LIN {X 0,Y 418.264,Z 439.007,A -85,B 0,C 180,E1 -10279.791,E2 -10279.791} C_VEL
LIN {X 0,Y 418.232,Z 439.016,A -85,B 0,C 180,E1 -10282.737,E2 -10282.737} C_VEL
LIN {X 0,Y 418.265,Z 439.008,A -85,B 0,C 180,E1 -10285.905,E2 -10285.905} C_VEL
LIN {X 0,Y 418.269,Z 439.007,A -85,B 0,C 180,E1 -10289.162,E2 -10289.162} C_VEL
LIN {X 0,Y 418.255,Z 439.008,A -85,B 0,C 180,E1 -10292.845,E2 -10292.845} C_VEL
LIN {X 0,Y 418.245,Z 439.015,A -85,B 0,C 180,E1 -10296.24,E2 -10296.24} C_VEL
LIN {X 0,Y 418.277,Z 439.018,A -85,B 0,C 180,E1 -10298.25,E2 -10298.25} C_VEL
LIN {X 0,Y 421.028,Z 450.162,A -85,B 0,C 180,E1 -10300.737,E2 -10300.737} C_VEL
LIN {X 0,Y 429.428,Z 469.629,A -85,B 0,C 180,E1 -10301.712,E2 -10301.712} C_VEL
LIN {X 0,Y 431.13,Z 477.405,A -85,B 0,C 180,E1 -10301.972,E2 -10301.972} C_VEL
LIN {X 0,Y 428.557,Z 614.749,A -85,B 0,C 180,E1 -10304.367,E2 -10304.367} C_VEL
LIN {X 0,Y 427.904,Z 630.406,A -85,B 0,C 180,E1 -10304.826,E2 -10304.826} C_VEL
LIN {X 0,Y 427.072,Z 645.206,A -85,B 0,C 180,E1 -10305.458,E2 -10305.458} C_VEL
LIN {X 0,Y 426.047,Z 660.031,A -85,B 0,C 180,E1 -10306.303,E2 -10306.303} C_VEL
LIN {X 0,Y 424.862,Z 673.816,A -85,B 0,C 180,E1 -10307.297,E2 -10307.297} C_VEL
LIN {X 0,Y 423.692,Z 686.587,A -85,B 0,C 180,E1 -10308.434,E2 -10308.434} C_VEL
LIN {X 0,Y 422.369,Z 699.367,A -85,B 0,C 180,E1 -10309.814,E2 -10309.814} C_VEL
LIN {X 0,Y 421.205,Z 710.398,A -85,B 0,C 180,E1 -10311.252,E2 -10311.252} C_VEL
LIN {X 0,Y 420.173,Z 719.587,A -85,B 0,C 180,E1 -10312.676,E2 -10312.676} C_VEL
LIN {X 0,Y 419.262,Z 728.801,A -85,B 0,C 180,E1 -10314.374,E2 -10314.374} C_VEL
LIN {X 0,Y 418.549,Z 736.533,A -85,B 0,C 180,E1 -10316.09,E2 -10316.09} C_VEL
LIN {X 0,Y 417.858,Z 743.619,A -85,B 0,C 180,E1 -10318.009,E2 -10318.009} C_VEL
LIN {X 0,Y 417.543,Z 748.582,A -85,B 0,C 180,E1 -10319.673,E2 -10319.673} C_VEL
LIN {X 0,Y 417.249,Z 752.105,A -85,B 0,C 180,E1 -10321.149,E2 -10321.149} C_VEL
LIN {X 0,Y 416.99,Z 755.939,A -85,B 0,C 180,E1 -10323.288,E2 -10323.288} C_VEL
LIN {X 0,Y 416.875,Z 758.426,A -85,B 0,C 180,E1 -10325.558,E2 -10325.558} C_VEL
LIN {X 0,Y 416.837,Z 759.366,A -85,B 0,C 180,E1 -10328.021,E2 -10328.021} C_VEL
LIN {X 0,Y 416.862,Z 758.566,A -85,B 0,C 180,E1 -10330.295,E2 -10330.295} C_VEL
LIN {X 0,Y 416.983,Z 756.515,A -85,B 0,C 180,E1 -10332.34,E2 -10332.34} C_VEL
LIN {X 0,Y 417.189,Z 753.759,A -85,B 0,C 180,E1 -10334.039,E2 -10334.039} C_VEL
LIN {X 0,Y 416.614,Z 752.269,A -85,B 0,C 180,E1 -10334.821,E2 -10334.821} C_VEL
LIN {X 0,Y 413.918,Z 749.553,A -85,B 0,C 180,E1 -10336.084,E2 -10336.084} C_VEL
LIN {X 0,Y 411.683,Z 747.027,A -85,B 0,C 180,E1 -10337.087,E2 -10337.087} C_VEL
LIN {X 0,Y 410.83,Z 744.837,A -85,B 0,C 180,E1 -10337.846,E2 -10337.846} C_VEL
LIN {X 0,Y 410.82,Z 744.026,A -85,B 0,C 180,E1 -10338.098,E2 -10338.098} C_VEL
LIN {X 0,Y 411.441,Z 736.535,A -85,B 0,C 180,E1 -10340.166,E2 -10340.166} C_VEL
LIN {X 0,Y 412.264,Z 728.503,A -85,B 0,C 180,E1 -10341.956,E2 -10341.956} C_VEL
LIN {X 0,Y 413.238,Z 719.329,A -85,B 0,C 180,E1 -10343.654,E2 -10343.654} C_VEL
LIN {X 0,Y 414.315,Z 709.798,A -85,B 0,C 180,E1 -10345.135,E2 -10345.135} C_VEL
LIN {X 0,Y 415.491,Z 698.732,A -85,B 0,C 180,E1 -10346.583,E2 -10346.583} C_VEL
LIN {X 0,Y 416.83,Z 686.135,A -85,B 0,C 180,E1 -10347.947,E2 -10347.947} C_VEL
LIN {X 0,Y 418.019,Z 674.003,A -85,B 0,C 180,E1 -10349.037,E2 -10349.037} C_VEL
LIN {X 0,Y 419.145,Z 660.909,A -85,B 0,C 180,E1 -10350.001,E2 -10350.001} C_VEL
LIN {X 0,Y 420.189,Z 646.609,A -85,B 0,C 180,E1 -10350.839,E2 -10350.839} C_VEL
LIN {X 0,Y 421.045,Z 631.881,A -85,B 0,C 180,E1 -10351.495,E2 -10351.495} C_VEL
LIN {X 0,Y 421.681,Z 616.76,A -85,B 0,C 180,E1 -10351.97,E2 -10351.97} C_VEL
LIN {X 0,Y 422.249,Z 590.391,A -85,B 0,C 180,E1 -10352.469,E2 -10352.469} C_VEL
LIN {X 0,Y 424.329,Z 477.84,A -85,B 0,C 180,E1 -10354.433,E2 -10354.433} C_VEL
LIN {X 0,Y 422.249,Z 469.646,A -85,B 0,C 180,E1 -10354.725,E2 -10354.725} C_VEL
LIN {X 0,Y 413.752,Z 449.749,A -85,B 0,C 180,E1 -10355.705,E2 -10355.705} C_VEL
LIN {X 0,Y 411.414,Z 439.866,A -85,B 0,C 180,E1 -10357.917,E2 -10357.917} C_VEL
LIN {X 0,Y 411.303,Z 439.874,A -85,B 0,C 180,E1 -10361.833,E2 -10361.833} C_VEL
LIN {X 0,Y 411.267,Z 439.881,A -85,B 0,C 180,E1 -10364.853,E2 -10364.853} C_VEL
LIN {X 0,Y 411.257,Z 439.88,A -85,B 0,C 180,E1 -10367.915,E2 -10367.915} C_VEL
LIN {X 0,Y 411.206,Z 439.885,A -85,B 0,C 180,E1 -10371.034,E2 -10371.034} C_VEL
LIN {X 0,Y 411.231,Z 439.879,A -85,B 0,C 180,E1 -10374.215,E2 -10374.215} C_VEL
LIN {X 0,Y 411.263,Z 439.878,A -85,B 0,C 180,E1 -10377.478,E2 -10377.478} C_VEL
LIN {X 0,Y 411.2,Z 439.888,A -85,B 0,C 180,E1 -10380.847,E2 -10380.847} C_VEL
LIN {X 0,Y 411.21,Z 439.886,A -85,B 0,C 180,E1 -10384.333,E2 -10384.333} C_VEL
LIN {X 0,Y 411.204,Z 439.879,A -85,B 0,C 180,E1 -10387.973,E2 -10387.973} C_VEL
LIN {X 0,Y 411.197,Z 439.889,A -85,B 0,C 180,E1 -10391.233,E2 -10391.233} C_VEL
LIN {X 0,Y 411.182,Z 439.887,A -85,B 0,C 180,E1 -10394.49,E2 -10394.49} C_VEL
LIN {X 0,Y 411.201,Z 439.879,A -85,B 0,C 180,E1 -10398.197,E2 -10398.197} C_VEL
LIN {X 0,Y 411.232,Z 439.882,A -85,B 0,C 180,E1 -10400.777,E2 -10400.777} C_VEL
LIN {X 0,Y 411.202,Z 439.879,A -85,B 0,C 180,E1 -10404.471,E2 -10404.471} C_VEL
LIN {X 0,Y 411.209,Z 439.885,A -85,B 0,C 180,E1 -10406.873,E2 -10406.873} C_VEL
LIN {X 0,Y 411.234,Z 439.873,A -85,B 0,C 180,E1 -10410.644,E2 -10410.644} C_VEL
LIN {X 0,Y 411.239,Z 439.888,A -85,B 0,C 180,E1 -10413.619,E2 -10413.619} C_VEL
LIN {X 0,Y 411.198,Z 439.874,A -85,B 0,C 180,E1 -10416.852,E2 -10416.852} C_VEL
LIN {X 0,Y 411.216,Z 439.886,A -85,B 0,C 180,E1 -10420.05,E2 -10420.05} C_VEL
LIN {X 0,Y 411.264,Z 439.871,A -85,B 0,C 180,E1 -10423.131,E2 -10423.131} C_VEL
LIN {X 0,Y 411.306,Z 439.872,A -85,B 0,C 180,E1 -10426.896,E2 -10426.896} C_VEL
LIN {X 0,Y 411.293,Z 439.865,A -85,B 0,C 180,E1 -10430.161,E2 -10430.161} C_VEL
LIN {X 0,Y 411.482,Z 439.851,A -85,B 0,C 180,E1 -10432.146,E2 -10432.146} C_VEL
LIN {X 0,Y 411.475,Z 439.853,A -85,B 0,C 180,E1 -10434.118,E2 -10434.118} C_VEL
LIN {X 0,Y 411.511,Z 439.845,A -85,B 0,C 180,E1 -10438.042,E2 -10438.042} C_VEL
LIN {X 0,Y 411.642,Z 439.835,A -85,B 0,C 180,E1 -10440,E2 -10440} C_VEL
LIN {X 0,Y 411.466,Z 439.848,A -85,B 0,C 180,E1 -10442.937,E2 -10442.937} C_VEL
LIN {X 0,Y 411.46,Z 439.85,A -85,B 0,C 180,E1 -10446.867,E2 -10446.867} C_VEL
LIN {X 0,Y 411.354,Z 439.867,A -85,B 0,C 180,E1 -10448.845,E2 -10448.845} C_VEL
LIN {X 0,Y 411.283,Z 439.866,A -85,B 0,C 180,E1 -10451.833,E2 -10451.833} C_VEL
LIN {X 0,Y 411.26,Z 439.878,A -85,B 0,C 180,E1 -10454.852,E2 -10454.852} C_VEL
LIN {X 0,Y 411.252,Z 439.871,A -85,B 0,C 180,E1 -10457.915,E2 -10457.915} C_VEL
LIN {X 0,Y 411.196,Z 439.886,A -85,B 0,C 180,E1 -10461.034,E2 -10461.034} C_VEL
LIN {X 0,Y 411.227,Z 439.885,A -85,B 0,C 180,E1 -10464.215,E2 -10464.215} C_VEL
LIN {X 0,Y 411.259,Z 439.883,A -85,B 0,C 180,E1 -10467.477,E2 -10467.477} C_VEL
LIN {X 0,Y 411.196,Z 439.885,A -85,B 0,C 180,E1 -10470.847,E2 -10470.847} C_VEL
LIN {X 0,Y 411.206,Z 439.887,A -85,B 0,C 180,E1 -10474.333,E2 -10474.333} C_VEL
LIN {X 0,Y 411.201,Z 439.889,A -85,B 0,C 180,E1 -10477.973,E2 -10477.973} C_VEL
LIN {X 0,Y 411.183,Z 439.889,A -85,B 0,C 180,E1 -10480.504,E2 -10480.504} C_VEL
LIN {X 0,Y 411.175,Z 439.891,A -85,B 0,C 180,E1 -10483.133,E2 -10483.133} C_VEL
LIN {X 0,Y 411.227,Z 439.886,A -85,B 0,C 180,E1 -10485.872,E2 -10485.872} C_VEL
LIN {X 0,Y 411.205,Z 439.888,A -85,B 0,C 180,E1 -10488.765,E2 -10488.765} C_VEL
LIN {X 0,Y 411.194,Z 439.892,A -85,B 0,C 180,E1 -10492.026,E2 -10492.026} C_VEL
LIN {X 0,Y 411.206,Z 439.887,A -85,B 0,C 180,E1 -10495.666,E2 -10495.666} C_VEL
LIN {X 0,Y 411.206,Z 439.954,A -85,B 0,C 180,E1 -10496.552,E2 -10496.552} C_VEL
LIN {X 0,Y 415.186,Z 455.473,A -85,B 0,C 180,E1 -10499.688,E2 -10499.688} C_VEL
LIN {X 0,Y 417.73,Z 467.012,A -85,B 0,C 180,E1 -10501.895,E2 -10501.895} C_VEL
LIN {X 0,Y 417.421,Z 471.137,A -85,B 0,C 180,E1 -10502.59,E2 -10502.59} C_VEL
LIN {X 0,Y 423.956,Z 504.652,A -85,B 0,C 180,E1 -10503.663,E2 -10503.663} C_VEL
LIN {X 0,Y 422.062,Z 609.761,A -85,B 0,C 180,E1 -10505.498,E2 -10505.498} C_VEL
LIN {X 0,Y 421.485,Z 639.304,A -85,B 0,C 180,E1 -10506.051,E2 -10506.051} C_VEL
LIN {X 0,Y 420.701,Z 654.425,A -85,B 0,C 180,E1 -10506.512,E2 -10506.512} C_VEL
LIN {X 0,Y 419.794,Z 669.444,A -85,B 0,C 180,E1 -10507.175,E2 -10507.175} C_VEL
LIN {X 0,Y 418.751,Z 682.833,A -85,B 0,C 180,E1 -10507.943,E2 -10507.943} C_VEL
LIN {X 0,Y 417.533,Z 696.274,A -85,B 0,C 180,E1 -10508.912,E2 -10508.912} C_VEL
LIN {X 0,Y 416.123,Z 709.958,A -85,B 0,C 180,E1 -10510.129,E2 -10510.129} C_VEL
LIN {X 0,Y 414.772,Z 722.886,A -85,B 0,C 180,E1 -10511.541,E2 -10511.541} C_VEL
LIN {X 0,Y 413.69,Z 733.682,A -85,B 0,C 180,E1 -10512.959,E2 -10512.959} C_VEL
LIN {X 0,Y 412.496,Z 744.676,A -85,B 0,C 180,E1 -10514.687,E2 -10514.687} C_VEL
LIN {X 0,Y 411.586,Z 753.834,A -85,B 0,C 180,E1 -10516.428,E2 -10516.428} C_VEL
LIN {X 0,Y 411.006,Z 761.372,A -85,B 0,C 180,E1 -10518.159,E2 -10518.159} C_VEL
LIN {X 0,Y 410.407,Z 768.44,A -85,B 0,C 180,E1 -10520.139,E2 -10520.139} C_VEL
LIN {X 0,Y 410.156,Z 774.002,A -85,B 0,C 180,E1 -10522.121,E2 -10522.121} C_VEL
LIN {X 0,Y 409.975,Z 778.206,A -85,B 0,C 180,E1 -10524.096,E2 -10524.096} C_VEL
LIN {X 0,Y 409.895,Z 781.155,A -85,B 0,C 180,E1 -10526.067,E2 -10526.067} C_VEL
LIN {X 0,Y 409.957,Z 782.918,A -85,B 0,C 180,E1 -10528.035,E2 -10528.035} C_VEL
LIN {X 0,Y 409.923,Z 783.517,A -85,B 0,C 180,E1 -10529.999,E2 -10529.999} C_VEL
LIN {X 0,Y 409.959,Z 782.915,A -85,B 0,C 180,E1 -10531.964,E2 -10531.964} C_VEL
LIN {X 0,Y 409.907,Z 781.16,A -85,B 0,C 180,E1 -10533.932,E2 -10533.932} C_VEL
LIN {X 0,Y 409.976,Z 778.229,A -85,B 0,C 180,E1 -10535.903,E2 -10535.903} C_VEL
LIN {X 0,Y 410.155,Z 774.051,A -85,B 0,C 180,E1 -10537.878,E2 -10537.878} C_VEL
LIN {X 0,Y 410.407,Z 768.515,A -85,B 0,C 180,E1 -10539.86,E2 -10539.86} C_VEL
LIN {X 0,Y 411.027,Z 761.48,A -85,B 0,C 180,E1 -10541.84,E2 -10541.84} C_VEL
LIN {X 0,Y 411.627,Z 753.862,A -85,B 0,C 180,E1 -10543.596,E2 -10543.596} C_VEL
LIN {X 0,Y 412.489,Z 744.879,A -85,B 0,C 180,E1 -10545.312,E2 -10545.312} C_VEL
LIN {X 0,Y 413.694,Z 733.993,A -85,B 0,C 180,E1 -10547.04,E2 -10547.04} C_VEL
LIN {X 0,Y 414.994,Z 722.266,A -85,B 0,C 180,E1 -10548.581,E2 -10548.581} C_VEL
LIN {X 0,Y 416.161,Z 710.536,A -85,B 0,C 180,E1 -10549.868,E2 -10549.868} C_VEL
LIN {X 0,Y 417.546,Z 697.077,A -85,B 0,C 180,E1 -10551.086,E2 -10551.086} C_VEL
LIN {X 0,Y 418.806,Z 683.881,A -85,B 0,C 180,E1 -10552.053,E2 -10552.053} C_VEL
LIN {X 0,Y 419.957,Z 669.116,A -85,B 0,C 180,E1 -10552.918,E2 -10552.918} C_VEL
LIN {X 0,Y 420.932,Z 654.325,A -85,B 0,C 180,E1 -10553.57,E2 -10553.57} C_VEL
LIN {X 0,Y 421.717,Z 639.333,A -85,B 0,C 180,E1 -10554.032,E2 -10554.032} C_VEL
LIN {X 0,Y 422.307,Z 613.685,A -85,B 0,C 180,E1 -10554.519,E2 -10554.519} C_VEL
LIN {X 0,Y 424.314,Z 504.605,A -85,B 0,C 180,E1 -10556.434,E2 -10556.434} C_VEL
LIN {X 0,Y 419.497,Z 479.497,A -85,B 0,C 180,E1 -10557.255,E2 -10557.255} C_VEL
LIN {X 0,Y 417.605,Z 470.44,A -85,B 0,C 180,E1 -10557.594,E2 -10557.594} C_VEL
LIN {X 0,Y 417.693,Z 466.142,A -85,B 0,C 180,E1 -10558.343,E2 -10558.343} C_VEL
LIN {X 0,Y 414.395,Z 451.915,A -85,B 0,C 180,E1 -10561.148,E2 -10561.148} C_VEL
LIN {X 0,Y 411.222,Z 439.886,A -85,B 0,C 180,E1 -10563.703,E2 -10563.703} C_VEL
LIN {X 0,Y 411.189,Z 439.89,A -85,B 0,C 180,E1 -10566.741,E2 -10566.741} C_VEL
LIN {X 0,Y 411.224,Z 439.882,A -85,B 0,C 180,E1 -10569.73,E2 -10569.73} C_VEL
LIN {X 0,Y 411.217,Z 439.881,A -85,B 0,C 180,E1 -10573.127,E2 -10573.127} C_VEL
LIN {X 0,Y 411.166,Z 439.891,A -85,B 0,C 180,E1 -10575.88,E2 -10575.88} C_VEL
LIN {X 0,Y 411.159,Z 439.895,A -85,B 0,C 180,E1 -10578.771,E2 -10578.771} C_VEL
LIN {X 0,Y 411.205,Z 439.888,A -85,B 0,C 180,E1 -10581.83,E2 -10581.83} C_VEL
LIN {X 0,Y 411.205,Z 439.887,A -85,B 0,C 180,E1 -10585.121,E2 -10585.121} C_VEL
LIN {X 0,Y 411.159,Z 439.893,A -85,B 0,C 180,E1 -10588.002,E2 -10588.002} C_VEL
LIN {X 0,Y 411.211,Z 439.886,A -85,B 0,C 180,E1 -10591.41,E2 -10591.41} C_VEL
LIN {X 0,Y 411.231,Z 439.88,A -85,B 0,C 180,E1 -10593.619,E2 -10593.619} C_VEL
LIN {X 0,Y 411.196,Z 439.889,A -85,B 0,C 180,E1 -10596.852,E2 -10596.852} C_VEL
LIN {X 0,Y 411.207,Z 439.884,A -85,B 0,C 180,E1 -10600.05,E2 -10600.05} C_VEL
LIN {X 0,Y 411.255,Z 439.875,A -85,B 0,C 180,E1 -10603.131,E2 -10603.131} C_VEL
LIN {X 0,Y 411.306,Z 439.871,A -85,B 0,C 180,E1 -10606.891,E2 -10606.891} C_VEL
LIN {X 0,Y 411.301,Z 439.874,A -85,B 0,C 180,E1 -10610.162,E2 -10610.162} C_VEL
LIN {X 0,Y 411.453,Z 439.853,A -85,B 0,C 180,E1 -10613.133,E2 -10613.133} C_VEL
LIN {X 0,Y 411.306,Z 439.873,A -85,B 0,C 180,E1 -10615.099,E2 -10615.099} C_VEL
LIN {X 0,Y 411.507,Z 439.846,A -85,B 0,C 180,E1 -10618.043,E2 -10618.043} C_VEL
LIN {X 0,Y 411.634,Z 439.836,A -85,B 0,C 180,E1 -10620,E2 -10620} C_VEL
LIN {X 0,Y 411.46,Z 439.856,A -85,B 0,C 180,E1 -10622.937,E2 -10622.937} C_VEL
LIN {X 0,Y 411.454,Z 439.856,A -85,B 0,C 180,E1 -10626.867,E2 -10626.867} C_VEL
LIN {X 0,Y 411.286,Z 439.878,A -85,B 0,C 180,E1 -10629.839,E2 -10629.839} C_VEL
LIN {X 0,Y 411.298,Z 439.874,A -85,B 0,C 180,E1 -10633.105,E2 -10633.105} C_VEL
LIN {X 0,Y 411.257,Z 439.882,A -85,B 0,C 180,E1 -10635.868,E2 -10635.868} C_VEL
LIN {X 0,Y 411.218,Z 439.885,A -85,B 0,C 180,E1 -10638.949,E2 -10638.949} C_VEL
LIN {X 0,Y 411.198,Z 439.894,A -85,B 0,C 180,E1 -10642.643,E2 -10642.643} C_VEL
LIN {X 0,Y 411.231,Z 439.886,A -85,B 0,C 180,E1 -10645.294,E2 -10645.294} C_VEL
LIN {X 0,Y 411.219,Z 439.89,A -85,B 0,C 180,E1 -10648.59,E2 -10648.59} C_VEL
LIN {X 0,Y 411.166,Z 439.893,A -85,B 0,C 180,E1 -10651.998,E2 -10651.998} C_VEL
LIN {X 0,Y 411.196,Z 439.891,A -85,B 0,C 180,E1 -10655.529,E2 -10655.529} C_VEL
LIN {X 0,Y 411.232,Z 439.979,A -85,B 0,C 180,E1 -10657.815,E2 -10657.815} C_VEL
LIN {X 0,Y 413.902,Z 450.487,A -85,B 0,C 180,E1 -10660.216,E2 -10660.216} C_VEL
LIN {X 0,Y 423.271,Z 471.849,A -85,B 0,C 180,E1 -10661.324,E2 -10661.324} C_VEL
LIN {X 0,Y 424.816,Z 478.598,A -85,B 0,C 180,E1 -10661.562,E2 -10661.562} C_VEL
LIN {X 0,Y 422.093,Z 615.228,A -85,B 0,C 180,E1 -10663.979,E2 -10663.979} C_VEL
LIN {X 0,Y 421.427,Z 630.771,A -85,B 0,C 180,E1 -10664.446,E2 -10664.446} C_VEL
LIN {X 0,Y 420.524,Z 645.75,A -85,B 0,C 180,E1 -10665.096,E2 -10665.096} C_VEL
LIN {X 0,Y 419.504,Z 659.931,A -85,B 0,C 180,E1 -10665.915,E2 -10665.915} C_VEL
LIN {X 0,Y 418.246,Z 674.101,A -85,B 0,C 180,E1 -10666.951,E2 -10666.951} C_VEL
LIN {X 0,Y 417,Z 686.839,A -85,B 0,C 180,E1 -10668.102,E2 -10668.102} C_VEL
LIN {X 0,Y 415.665,Z 699.15,A -85,B 0,C 180,E1 -10669.449,E2 -10669.449} C_VEL
LIN {X 0,Y 414.504,Z 709.69,A -85,B 0,C 180,E1 -10670.834,E2 -10670.834} C_VEL
LIN {X 0,Y 413.254,Z 720.367,A -85,B 0,C 180,E1 -10672.504,E2 -10672.504} C_VEL
LIN {X 0,Y 412.246,Z 729.718,A -85,B 0,C 180,E1 -10674.276,E2 -10674.276} C_VEL
LIN {X 0,Y 411.516,Z 737.209,A -85,B 0,C 180,E1 -10675.993,E2 -10675.993} C_VEL
LIN {X 0,Y 410.806,Z 744.291,A -85,B 0,C 180,E1 -10677.972,E2 -10677.972} C_VEL
LIN {X 0,Y 410.46,Z 749.144,A -85,B 0,C 180,E1 -10679.663,E2 -10679.663} C_VEL
LIN {X 0,Y 410.052,Z 754.007,A -85,B 0,C 180,E1 -10681.88,E2 -10681.88} C_VEL
LIN {X 0,Y 409.882,Z 756.625,A -85,B 0,C 180,E1 -10683.526,E2 -10683.526} C_VEL
LIN {X 0,Y 409.776,Z 758.784,A -85,B 0,C 180,E1 -10685.694,E2 -10685.694} C_VEL
LIN {X 0,Y 409.727,Z 759.555,A -85,B 0,C 180,E1 -10687.859,E2 -10687.859} C_VEL
LIN {X 0,Y 409.756,Z 758.996,A -85,B 0,C 180,E1 -10689.939,E2 -10689.939} C_VEL
LIN {X 0,Y 409.855,Z 757.165,A -85,B 0,C 180,E1 -10692.023,E2 -10692.023} C_VEL
LIN {X 0,Y 410.12,Z 754.049,A -85,B 0,C 180,E1 -10694.087,E2 -10694.087} C_VEL
LIN {X 0,Y 410.409,Z 749.635,A -85,B 0,C 180,E1 -10696.129,E2 -10696.129} C_VEL
LIN {X 0,Y 410.82,Z 744.026,A -85,B 0,C 180,E1 -10698.098,E2 -10698.098} C_VEL
LIN {X 0,Y 410.391,Z 741.613,A -85,B 0,C 180,E1 -10698.847,E2 -10698.847} C_VEL
LIN {X 0,Y 407.957,Z 737.47,A -85,B 0,C 180,E1 -10700.064,E2 -10700.064} C_VEL
LIN {X 0,Y 405.567,Z 732.91,A -85,B 0,C 180,E1 -10701.261,E2 -10701.261} C_VEL
LIN {X 0,Y 405.21,Z 729.776,A -85,B 0,C 180,E1 -10701.969,E2 -10701.969} C_VEL
LIN {X 0,Y 406.128,Z 721.688,A -85,B 0,C 180,E1 -10703.542,E2 -10703.542} C_VEL
LIN {X 0,Y 407.399,Z 710.839,A -85,B 0,C 180,E1 -10705.3,E2 -10705.3} C_VEL
LIN {X 0,Y 408.736,Z 698.783,A -85,B 0,C 180,E1 -10706.907,E2 -10706.907} C_VEL
LIN {X 0,Y 410.114,Z 686.258,A -85,B 0,C 180,E1 -10708.282,E2 -10708.282} C_VEL
LIN {X 0,Y 411.357,Z 674.103,A -85,B 0,C 180,E1 -10709.389,E2 -10709.389} C_VEL
LIN {X 0,Y 412.539,Z 660.969,A -85,B 0,C 180,E1 -10710.367,E2 -10710.367} C_VEL
LIN {X 0,Y 413.632,Z 646.613,A -85,B 0,C 180,E1 -10711.218,E2 -10711.218} C_VEL
LIN {X 0,Y 414.541,Z 631.793,A -85,B 0,C 180,E1 -10711.883,E2 -10711.883} C_VEL
LIN {X 0,Y 415.203,Z 616.687,A -85,B 0,C 180,E1 -10712.36,E2 -10712.36} C_VEL
LIN {X 0,Y 415.784,Z 589.807,A -85,B 0,C 180,E1 -10712.874,E2 -10712.874} C_VEL
LIN {X 0,Y 417.916,Z 478.938,A -85,B 0,C 180,E1 -10714.84,E2 -10714.84} C_VEL
LIN {X 0,Y 416.032,Z 471.89,A -85,B 0,C 180,E1 -10715.104,E2 -10715.104} C_VEL
LIN {X 0,Y 406.578,Z 449.9,A -85,B 0,C 180,E1 -10716.234,E2 -10716.234} C_VEL
LIN {X 0,Y 404.364,Z 440.742,A -85,B 0,C 180,E1 -10718.332,E2 -10718.332} C_VEL
LIN {X 0,Y 404.274,Z 440.752,A -85,B 0,C 180,E1 -10722.041,E2 -10722.041} C_VEL
LIN {X 0,Y 404.212,Z 440.761,A -85,B 0,C 180,E1 -10725.118,E2 -10725.118} C_VEL
LIN {X 0,Y 404.218,Z 440.757,A -85,B 0,C 180,E1 -10728.238,E2 -10728.238} C_VEL
LIN {X 0,Y 404.146,Z 440.766,A -85,B 0,C 180,E1 -10731.419,E2 -10731.419} C_VEL
LIN {X 0,Y 404.181,Z 440.756,A -85,B 0,C 180,E1 -10734.666,E2 -10734.666} C_VEL
LIN {X 0,Y 404.201,Z 440.754,A -85,B 0,C 180,E1 -10738,E2 -10738} C_VEL
LIN {X 0,Y 404.146,Z 440.765,A -85,B 0,C 180,E1 -10741.559,E2 -10741.559} C_VEL
LIN {X 0,Y 404.189,Z 440.761,A -85,B 0,C 180,E1 -10745.016,E2 -10745.016} C_VEL
LIN {X 0,Y 404.162,Z 440.755,A -85,B 0,C 180,E1 -10748.756,E2 -10748.756} C_VEL
LIN {X 0,Y 404.144,Z 440.769,A -85,B 0,C 180,E1 -10751.603,E2 -10751.603} C_VEL
LIN {X 0,Y 404.151,Z 440.763,A -85,B 0,C 180,E1 -10754.522,E2 -10754.522} C_VEL
LIN {X 0,Y 404.173,Z 440.764,A -85,B 0,C 180,E1 -10757.3,E2 -10757.3} C_VEL
LIN {X 0,Y 404.171,Z 440.765,A -85,B 0,C 180,E1 -10759.955,E2 -10759.955} C_VEL
LIN {X 0,Y 404.142,Z 440.764,A -85,B 0,C 180,E1 -10763.124,E2 -10763.124} C_VEL
LIN {X 0,Y 404.147,Z 440.766,A -85,B 0,C 180,E1 -10766.188,E2 -10766.188} C_VEL
LIN {X 0,Y 404.147,Z 440.759,A -85,B 0,C 180,E1 -10769.715,E2 -10769.715} C_VEL
LIN {X 0,Y 404.196,Z 440.759,A -85,B 0,C 180,E1 -10773.123,E2 -10773.123} C_VEL
LIN {X 0,Y 404.176,Z 440.762,A -85,B 0,C 180,E1 -10775.334,E2 -10775.334} C_VEL
LIN {X 0,Y 404.139,Z 440.763,A -85,B 0,C 180,E1 -10778.58,E2 -10778.58} C_VEL
LIN {X 0,Y 404.211,Z 440.754,A -85,B 0,C 180,E1 -10781.762,E2 -10781.762} C_VEL
LIN {X 0,Y 404.207,Z 440.751,A -85,B 0,C 180,E1 -10784.882,E2 -10784.882} C_VEL
LIN {X 0,Y 404.257,Z 440.75,A -85,B 0,C 180,E1 -10787.958,E2 -10787.958} C_VEL
LIN {X 0,Y 404.434,Z 440.73,A -85,B 0,C 180,E1 -10792.099,E2 -10792.099} C_VEL
LIN {X 0,Y 404.424,Z 440.732,A -85,B 0,C 180,E1 -10794.015,E2 -10794.015} C_VEL
LIN {X 0,Y 404.48,Z 440.719,A -85,B 0,C 180,E1 -10798.008,E2 -10798.008} C_VEL
LIN {X 0,Y 404.611,Z 440.71,A -85,B 0,C 180,E1 -10800,E2 -10800} C_VEL
LIN {X 0,Y 404.422,Z 440.726,A -85,B 0,C 180,E1 -10802.988,E2 -10802.988} C_VEL
LIN {X 0,Y 404.411,Z 440.728,A -85,B 0,C 180,E1 -10806.987,E2 -10806.987} C_VEL
LIN {X 0,Y 404.258,Z 440.748,A -85,B 0,C 180,E1 -10810.011,E2 -10810.011} C_VEL
LIN {X 0,Y 404.266,Z 440.741,A -85,B 0,C 180,E1 -10813.211,E2 -10813.211} C_VEL
LIN {X 0,Y 404.216,Z 440.755,A -85,B 0,C 180,E1 -10817.007,E2 -10817.007} C_VEL
LIN {X 0,Y 404.163,Z 440.763,A -85,B 0,C 180,E1 -10820.351,E2 -10820.351} C_VEL
LIN {X 0,Y 404.169,Z 440.765,A -85,B 0,C 180,E1 -10823.574,E2 -10823.574} C_VEL
LIN {X 0,Y 404.184,Z 440.763,A -85,B 0,C 180,E1 -10825.766,E2 -10825.766} C_VEL
LIN {X 0,Y 404.196,Z 440.76,A -85,B 0,C 180,E1 -10827.999,E2 -10827.999} C_VEL
LIN {X 0,Y 404.142,Z 440.768,A -85,B 0,C 180,E1 -10831.558,E2 -10831.558} C_VEL
LIN {X 0,Y 404.185,Z 440.761,A -85,B 0,C 180,E1 -10835.016,E2 -10835.016} C_VEL
LIN {X 0,Y 404.159,Z 440.763,A -85,B 0,C 180,E1 -10838.756,E2 -10838.756} C_VEL
LIN {X 0,Y 404.124,Z 440.774,A -85,B 0,C 180,E1 -10841.6,E2 -10841.6} C_VEL
LIN {X 0,Y 404.154,Z 440.765,A -85,B 0,C 180,E1 -10844.523,E2 -10844.523} C_VEL
LIN {X 0,Y 404.206,Z 440.762,A -85,B 0,C 180,E1 -10847.305,E2 -10847.305} C_VEL
LIN {X 0,Y 404.169,Z 440.766,A -85,B 0,C 180,E1 -10849.955,E2 -10849.955} C_VEL
LIN {X 0,Y 404.136,Z 440.765,A -85,B 0,C 180,E1 -10853.125,E2 -10853.125} C_VEL
LIN {X 0,Y 404.19,Z 440.822,A -85,B 0,C 180,E1 -10856.117,E2 -10856.117} C_VEL
LIN {X 0,Y 408.249,Z 456.728,A -85,B 0,C 180,E1 -10859.4,E2 -10859.4} C_VEL
LIN {X 0,Y 410.845,Z 468.295,A -85,B 0,C 180,E1 -10861.66,E2 -10861.66} C_VEL
LIN {X 0,Y 410.848,Z 471.29,A -85,B 0,C 180,E1 -10862.139,E2 -10862.139} C_VEL
LIN {X 0,Y 417.556,Z 505.795,A -85,B 0,C 180,E1 -10863.266,E2 -10863.266} C_VEL
LIN {X 0,Y 415.081,Z 635.987,A -85,B 0,C 180,E1 -10865.591,E2 -10865.591} C_VEL
LIN {X 0,Y 414.363,Z 651.574,A -85,B 0,C 180,E1 -10866.039,E2 -10866.039} C_VEL
LIN {X 0,Y 413.44,Z 665.662,A -85,B 0,C 180,E1 -10866.626,E2 -10866.626} C_VEL
LIN {X 0,Y 412.444,Z 678.457,A -85,B 0,C 180,E1 -10867.323,E2 -10867.323} C_VEL
LIN {X 0,Y 411.143,Z 692.736,A -85,B 0,C 180,E1 -10868.305,E2 -10868.305} C_VEL
LIN {X 0,Y 409.843,Z 705.752,A -85,B 0,C 180,E1 -10869.418,E2 -10869.418} C_VEL
LIN {X 0,Y 408.507,Z 717.775,A -85,B 0,C 180,E1 -10870.659,E2 -10870.659} C_VEL
LIN {X 0,Y 407.446,Z 727.998,A -85,B 0,C 180,E1 -10871.911,E2 -10871.911} C_VEL
LIN {X 0,Y 406.226,Z 738.36,A -85,B 0,C 180,E1 -10873.413,E2 -10873.413} C_VEL
LIN {X 0,Y 405.137,Z 748.516,A -85,B 0,C 180,E1 -10875.174,E2 -10875.174} C_VEL
LIN {X 0,Y 404.206,Z 756.946,A -85,B 0,C 180,E1 -10876.936,E2 -10876.936} C_VEL
LIN {X 0,Y 403.678,Z 764.867,A -85,B 0,C 180,E1 -10878.959,E2 -10878.959} C_VEL
LIN {X 0,Y 403.203,Z 771.166,A -85,B 0,C 180,E1 -10880.974,E2 -10880.974} C_VEL
LIN {X 0,Y 402.981,Z 776.041,A -85,B 0,C 180,E1 -10882.987,E2 -10882.987} C_VEL
LIN {X 0,Y 402.874,Z 779.615,A -85,B 0,C 180,E1 -10884.996,E2 -10884.996} C_VEL
LIN {X 0,Y 402.799,Z 781.968,A -85,B 0,C 180,E1 -10886.999,E2 -10886.999} C_VEL
LIN {X 0,Y 402.859,Z 783.157,A -85,B 0,C 180,E1 -10889,E2 -10889} C_VEL
LIN {X 0,Y 402.859,Z 783.153,A -85,B 0,C 180,E1 -10890.999,E2 -10890.999} C_VEL
LIN {X 0,Y 402.807,Z 781.978,A -85,B 0,C 180,E1 -10893,E2 -10893} C_VEL
LIN {X 0,Y 402.875,Z 779.646,A -85,B 0,C 180,E1 -10895.003,E2 -10895.003} C_VEL
LIN {X 0,Y 402.986,Z 776.104,A -85,B 0,C 180,E1 -10897.011,E2 -10897.011} C_VEL
LIN {X 0,Y 403.209,Z 771.266,A -85,B 0,C 180,E1 -10899.025,E2 -10899.025} C_VEL
LIN {X 0,Y 403.676,Z 765.004,A -85,B 0,C 180,E1 -10901.04,E2 -10901.04} C_VEL
LIN {X 0,Y 404.216,Z 757.14,A -85,B 0,C 180,E1 -10903.063,E2 -10903.063} C_VEL
LIN {X 0,Y 405.133,Z 748.793,A -85,B 0,C 180,E1 -10904.825,E2 -10904.825} C_VEL
LIN {X 0,Y 406.211,Z 738.746,A -85,B 0,C 180,E1 -10906.586,E2 -10906.586} C_VEL
LIN {X 0,Y 407.615,Z 727.252,A -85,B 0,C 180,E1 -10908.249,E2 -10908.249} C_VEL
LIN {X 0,Y 408.897,Z 715.112,A -85,B 0,C 180,E1 -10909.712,E2 -10909.712} C_VEL
LIN {X 0,Y 410.335,Z 702.679,A -85,B 0,C 180,E1 -10910.948,E2 -10910.948} C_VEL
LIN {X 0,Y 411.69,Z 689.081,A -85,B 0,C 180,E1 -10912.058,E2 -10912.058} C_VEL
LIN {X 0,Y 412.969,Z 675.027,A -85,B 0,C 180,E1 -10912.976,E2 -10912.976} C_VEL
LIN {X 0,Y 414.113,Z 659.618,A -85,B 0,C 180,E1 -10913.75,E2 -10913.75} C_VEL
LIN {X 0,Y 415.017,Z 645.021,A -85,B 0,C 180,E1 -10914.278,E2 -10914.278} C_VEL
LIN {X 0,Y 415.57,Z 629.766,A -85,B 0,C 180,E1 -10914.643,E2 -10914.643} C_VEL
LIN {X 0,Y 418.048,Z 506.433,A -85,B 0,C 180,E1 -10916.838,E2 -10916.838} C_VEL
LIN {X 0,Y 413.372,Z 481.506,A -85,B 0,C 180,E1 -10917.665,E2 -10917.665} C_VEL
LIN {X 0,Y 410.995,Z 470.32,A -85,B 0,C 180,E1 -10918.077,E2 -10918.077} C_VEL
LIN {X 0,Y 410.795,Z 467.367,A -85,B 0,C 180,E1 -10918.621,E2 -10918.621} C_VEL
LIN {X 0,Y 407.6,Z 453.661,A -85,B 0,C 180,E1 -10921.385,E2 -10921.385} C_VEL
LIN {X 0,Y 404.182,Z 440.767,A -85,B 0,C 180,E1 -10924.183,E2 -10924.183} C_VEL
LIN {X 0,Y 404.145,Z 440.764,A -85,B 0,C 180,E1 -10927.49,E2 -10927.49} C_VEL
LIN {X 0,Y 404.163,Z 440.761,A -85,B 0,C 180,E1 -10930.083,E2 -10930.083} C_VEL
LIN {X 0,Y 404.192,Z 440.755,A -85,B 0,C 180,E1 -10933.09,E2 -10933.09} C_VEL
LIN {X 0,Y 404.146,Z 440.764,A -85,B 0,C 180,E1 -10935.926,E2 -10935.926} C_VEL
LIN {X 0,Y 404.114,Z 440.774,A -85,B 0,C 180,E1 -10938.634,E2 -10938.634} C_VEL
LIN {X 0,Y 404.152,Z 440.766,A -85,B 0,C 180,E1 -10941.491,E2 -10941.491} C_VEL
LIN {X 0,Y 404.179,Z 440.762,A -85,B 0,C 180,E1 -10944.984,E2 -10944.984} C_VEL
LIN {X 0,Y 404.135,Z 440.77,A -85,B 0,C 180,E1 -10948.553,E2 -10948.553} C_VEL
LIN {X 0,Y 404.188,Z 440.764,A -85,B 0,C 180,E1 -10952,E2 -10952} C_VEL
LIN {X 0,Y 404.17,Z 440.762,A -85,B 0,C 180,E1 -10955.334,E2 -10955.334} C_VEL
LIN {X 0,Y 404.131,Z 440.768,A -85,B 0,C 180,E1 -10958.58,E2 -10958.58} C_VEL
LIN {X 0,Y 404.203,Z 440.76,A -85,B 0,C 180,E1 -10961.762,E2 -10961.762} C_VEL
LIN {X 0,Y 404.2,Z 440.76,A -85,B 0,C 180,E1 -10964.882,E2 -10964.882} C_VEL
LIN {X 0,Y 404.262,Z 440.75,A -85,B 0,C 180,E1 -10967.959,E2 -10967.959} C_VEL
LIN {X 0,Y 404.426,Z 440.733,A -85,B 0,C 180,E1 -10972.1,E2 -10972.1} C_VEL
LIN {X 0,Y 404.416,Z 440.73,A -85,B 0,C 180,E1 -10974.015,E2 -10974.015} C_VEL
LIN {X 0,Y 404.476,Z 440.722,A -85,B 0,C 180,E1 -10978.009,E2 -10978.009} C_VEL
LIN {X 0,Y 404.604,Z 440.711,A -85,B 0,C 180,E1 -10980,E2 -10980} C_VEL
LIN {X 0,Y 404.418,Z 440.733,A -85,B 0,C 180,E1 -10982.989,E2 -10982.989} C_VEL
LIN {X 0,Y 404.405,Z 440.733,A -85,B 0,C 180,E1 -10986.988,E2 -10986.988} C_VEL
LIN {X 0,Y 404.252,Z 440.756,A -85,B 0,C 180,E1 -10990.012,E2 -10990.012} C_VEL
LIN {X 0,Y 404.259,Z 440.751,A -85,B 0,C 180,E1 -10993.212,E2 -10993.212} C_VEL
LIN {X 0,Y 404.212,Z 440.759,A -85,B 0,C 180,E1 -10997.009,E2 -10997.009} C_VEL
LIN {X 0,Y 404.181,Z 440.767,A -85,B 0,C 180,E1 -11000.351,E2 -11000.351} C_VEL
LIN {X 0,Y 404.164,Z 440.766,A -85,B 0,C 180,E1 -11003.575,E2 -11003.575} C_VEL
LIN {X 0,Y 404.178,Z 440.764,A -85,B 0,C 180,E1 -11005.767,E2 -11005.767} C_VEL
LIN {X 0,Y 404.193,Z 440.764,A -85,B 0,C 180,E1 -11008,E2 -11008} C_VEL
LIN {X 0,Y 404.141,Z 440.769,A -85,B 0,C 180,E1 -11011.56,E2 -11011.56} C_VEL
LIN {X 0,Y 404.181,Z 440.761,A -85,B 0,C 180,E1 -11015.017,E2 -11015.017} C_VEL
LIN {X 0,Y 404.163,Z 440.876,A -85,B 0,C 180,E1 -11017.346,E2 -11017.346} C_VEL
LIN {X 0,Y 406.749,Z 450.708,A -85,B 0,C 180,E1 -11019.66,E2 -11019.66} C_VEL
LIN {X 0,Y 416.377,Z 472.267,A -85,B 0,C 180,E1 -11020.832,E2 -11020.832} C_VEL
LIN {X 0,Y 417.72,Z 476.244,A -85,B 0,C 180,E1 -11021.008,E2 -11021.008} C_VEL
LIN {X 0,Y 418.472,Z 480.588,A -85,B 0,C 180,E1 -11021.147,E2 -11021.147} C_VEL
LIN {X 0,Y 415.655,Z 615.446,A -85,B 0,C 180,E1 -11023.574,E2 -11023.574} C_VEL
LIN {X 0,Y 414.955,Z 630.729,A -85,B 0,C 180,E1 -11024.035,E2 -11024.035} C_VEL
LIN {X 0,Y 414.133,Z 644.371,A -85,B 0,C 180,E1 -11024.629,E2 -11024.629} C_VEL
LIN {X 0,Y 413.082,Z 658.448,A -85,B 0,C 180,E1 -11025.43,E2 -11025.43} C_VEL
LIN {X 0,Y 411.813,Z 672.55,A -85,B 0,C 180,E1 -11026.447,E2 -11026.447} C_VEL
LIN {X 0,Y 410.505,Z 685.458,A -85,B 0,C 180,E1 -11027.601,E2 -11027.601} C_VEL
LIN {X 0,Y 409.117,Z 697.684,A -85,B 0,C 180,E1 -11028.925,E2 -11028.925} C_VEL
LIN {X 0,Y 407.823,Z 708.896,A -85,B 0,C 180,E1 -11030.387,E2 -11030.387} C_VEL
LIN {X 0,Y 406.626,Z 718.312,A -85,B 0,C 180,E1 -11031.839,E2 -11031.839} C_VEL
LIN {X 0,Y 405.578,Z 727.826,A -85,B 0,C 180,E1 -11033.596,E2 -11033.596} C_VEL
LIN {X 0,Y 404.657,Z 735.686,A -85,B 0,C 180,E1 -11035.335,E2 -11035.335} C_VEL
LIN {X 0,Y 404.055,Z 741.819,A -85,B 0,C 180,E1 -11036.966,E2 -11036.966} C_VEL
LIN {X 0,Y 403.48,Z 748.343,A -85,B 0,C 180,E1 -11039.109,E2 -11039.109} C_VEL
LIN {X 0,Y 403.155,Z 752.299,A -85,B 0,C 180,E1 -11040.785,E2 -11040.785} C_VEL
LIN {X 0,Y 402.827,Z 756.243,A -85,B 0,C 180,E1 -11043.025,E2 -11043.025} C_VEL
LIN {X 0,Y 402.717,Z 758.673,A -85,B 0,C 180,E1 -11045.24,E2 -11045.24} C_VEL
LIN {X 0,Y 402.645,Z 759.698,A -85,B 0,C 180,E1 -11047.419,E2 -11047.419} C_VEL
LIN {X 0,Y 402.66,Z 759.393,A -85,B 0,C 180,E1 -11049.57,E2 -11049.57} C_VEL
LIN {X 0,Y 402.744,Z 757.808,A -85,B 0,C 180,E1 -11051.694,E2 -11051.694} C_VEL
LIN {X 0,Y 403.002,Z 754.942,A -85,B 0,C 180,E1 -11053.799,E2 -11053.799} C_VEL
LIN {X 0,Y 403.292,Z 750.782,A -85,B 0,C 180,E1 -11055.88,E2 -11055.88} C_VEL
LIN {X 0,Y 403.693,Z 745.264,A -85,B 0,C 180,E1 -11057.942,E2 -11057.942} C_VEL
LIN {X 0,Y 404.365,Z 738.234,A -85,B 0,C 180,E1 -11059.992,E2 -11059.992} C_VEL
LIN {X 0,Y 405.21,Z 729.776,A -85,B 0,C 180,E1 -11061.969,E2 -11061.969} C_VEL
LIN {X 0,Y 404.901,Z 726.52,A -85,B 0,C 180,E1 -11062.664,E2 -11062.664} C_VEL
LIN {X 0,Y 402.765,Z 721.087,A -85,B 0,C 180,E1 -11063.803,E2 -11063.803} C_VEL
LIN {X 0,Y 400.709,Z 715.256,A -85,B 0,C 180,E1 -11064.908,E2 -11064.908} C_VEL
LIN {X 0,Y 400.52,Z 711.345,A -85,B 0,C 180,E1 -11065.54,E2 -11065.54} C_VEL
LIN {X 0,Y 401.88,Z 699.828,A -85,B 0,C 180,E1 -11067.119,E2 -11067.119} C_VEL
LIN {X 0,Y 403.288,Z 687.605,A -85,B 0,C 180,E1 -11068.503,E2 -11068.503} C_VEL
LIN {X 0,Y 404.736,Z 674.173,A -85,B 0,C 180,E1 -11069.752,E2 -11069.752} C_VEL
LIN {X 0,Y 405.971,Z 661.007,A -85,B 0,C 180,E1 -11070.744,E2 -11070.744} C_VEL
LIN {X 0,Y 407.083,Z 646.629,A -85,B 0,C 180,E1 -11071.608,E2 -11071.608} C_VEL
LIN {X 0,Y 408.072,Z 630.699,A -85,B 0,C 180,E1 -11072.326,E2 -11072.326} C_VEL
LIN {X 0,Y 408.785,Z 615.236,A -85,B 0,C 180,E1 -11072.8,E2 -11072.8} C_VEL
LIN {X 0,Y 411.519,Z 480.305,A -85,B 0,C 180,E1 -11075.254,E2 -11075.254} C_VEL
LIN {X 0,Y 410.051,Z 474.685,A -85,B 0,C 180,E1 -11075.467,E2 -11075.467} C_VEL
LIN {X 0,Y 399.385,Z 450.144,A -85,B 0,C 180,E1 -11076.762,E2 -11076.762} C_VEL
LIN {X 0,Y 397.282,Z 441.625,A -85,B 0,C 180,E1 -11078.738,E2 -11078.738} C_VEL
LIN {X 0,Y 397.233,Z 441.632,A -85,B 0,C 180,E1 -11082.258,E2 -11082.258} C_VEL
LIN {X 0,Y 397.184,Z 441.634,A -85,B 0,C 180,E1 -11085.392,E2 -11085.392} C_VEL
LIN {X 0,Y 397.175,Z 441.634,A -85,B 0,C 180,E1 -11088.573,E2 -11088.573} C_VEL
LIN {X 0,Y 397.103,Z 441.646,A -85,B 0,C 180,E1 -11091.818,E2 -11091.818} C_VEL
LIN {X 0,Y 397.161,Z 441.633,A -85,B 0,C 180,E1 -11095.132,E2 -11095.132} C_VEL
LIN {X 0,Y 397.167,Z 441.631,A -85,B 0,C 180,E1 -11097.776,E2 -11097.776} C_VEL
LIN {X 0,Y 397.087,Z 441.646,A -85,B 0,C 180,E1 -11100.882,E2 -11100.882} C_VEL
LIN {X 0,Y 397.129,Z 441.64,A -85,B 0,C 180,E1 -11104.493,E2 -11104.493} C_VEL
LIN {X 0,Y 397.11,Z 441.634,A -85,B 0,C 180,E1 -11108.274,E2 -11108.274} C_VEL
LIN {X 0,Y 397.11,Z 441.642,A -85,B 0,C 180,E1 -11110.906,E2 -11110.906} C_VEL
LIN {X 0,Y 397.106,Z 441.639,A -85,B 0,C 180,E1 -11113.648,E2 -11113.648} C_VEL
LIN {X 0,Y 397.106,Z 441.641,A -85,B 0,C 180,E1 -11116.52,E2 -11116.52} C_VEL
LIN {X 0,Y 397.122,Z 441.637,A -85,B 0,C 180,E1 -11119.551,E2 -11119.551} C_VEL
LIN {X 0,Y 397.101,Z 441.64,A -85,B 0,C 180,E1 -11122.79,E2 -11122.79} C_VEL
LIN {X 0,Y 397.12,Z 441.641,A -85,B 0,C 180,E1 -11126.282,E2 -11126.282} C_VEL
LIN {X 0,Y 397.106,Z 441.634,A -85,B 0,C 180,E1 -11130.135,E2 -11130.135} C_VEL
LIN {X 0,Y 397.196,Z 441.63,A -85,B 0,C 180,E1 -11132.61,E2 -11132.61} C_VEL
LIN {X 0,Y 397.13,Z 441.629,A -85,B 0,C 180,E1 -11135.981,E2 -11135.981} C_VEL
LIN {X 0,Y 397.14,Z 441.643,A -85,B 0,C 180,E1 -11139.704,E2 -11139.704} C_VEL
LIN {X 0,Y 397.183,Z 441.623,A -85,B 0,C 180,E1 -11142.845,E2 -11142.845} C_VEL
LIN {X 0,Y 397.229,Z 441.626,A -85,B 0,C 180,E1 -11146.702,E2 -11146.702} C_VEL
LIN {X 0,Y 397.218,Z 441.619,A -85,B 0,C 180,E1 -11149.809,E2 -11149.809} C_VEL
LIN {X 0,Y 397.364,Z 441.608,A -85,B 0,C 180,E1 -11152.888,E2 -11152.888} C_VEL
LIN {X 0,Y 397.255,Z 441.622,A -85,B 0,C 180,E1 -11154.925,E2 -11154.925} C_VEL
LIN {X 0,Y 397.449,Z 441.594,A -85,B 0,C 180,E1 -11157.973,E2 -11157.973} C_VEL
LIN {X 0,Y 397.581,Z 441.586,A -85,B 0,C 180,E1 -11160,E2 -11160} C_VEL
LIN {X 0,Y 397.381,Z 441.603,A -85,B 0,C 180,E1 -11163.041,E2 -11163.041} C_VEL
LIN {X 0,Y 397.364,Z 441.607,A -85,B 0,C 180,E1 -11167.112,E2 -11167.112} C_VEL
LIN {X 0,Y 397.218,Z 441.623,A -85,B 0,C 180,E1 -11170.191,E2 -11170.191} C_VEL
LIN {X 0,Y 397.226,Z 441.619,A -85,B 0,C 180,E1 -11173.321,E2 -11173.321} C_VEL
LIN {X 0,Y 397.182,Z 441.632,A -85,B 0,C 180,E1 -11177.155,E2 -11177.155} C_VEL
LIN {X 0,Y 397.102,Z 441.641,A -85,B 0,C 180,E1 -11180.73,E2 -11180.73} C_VEL
LIN {X 0,Y 397.133,Z 441.642,A -85,B 0,C 180,E1 -11184.018,E2 -11184.018} C_VEL
LIN {X 0,Y 397.194,Z 441.634,A -85,B 0,C 180,E1 -11187.39,E2 -11187.39} C_VEL
LIN {X 0,Y 397.083,Z 441.643,A -85,B 0,C 180,E1 -11190.882,E2 -11190.882} C_VEL
LIN {X 0,Y 397.126,Z 441.64,A -85,B 0,C 180,E1 -11194.493,E2 -11194.493} C_VEL
LIN {X 0,Y 397.107,Z 441.643,A -85,B 0,C 180,E1 -11198.274,E2 -11198.274} C_VEL
LIN {X 0,Y 397.089,Z 441.644,A -85,B 0,C 180,E1 -11200.908,E2 -11200.908} C_VEL
LIN {X 0,Y 397.103,Z 441.648,A -85,B 0,C 180,E1 -11203.648,E2 -11203.648} C_VEL
LIN {X 0,Y 397.159,Z 441.637,A -85,B 0,C 180,E1 -11206.512,E2 -11206.512} C_VEL
LIN {X 0,Y 397.115,Z 441.644,A -85,B 0,C 180,E1 -11209.552,E2 -11209.552} C_VEL
LIN {X 0,Y 397.094,Z 441.644,A -85,B 0,C 180,E1 -11212.791,E2 -11212.791} C_VEL
LIN {X 0,Y 397.124,Z 441.669,A -85,B 0,C 180,E1 -11215.661,E2 -11215.661} C_VEL
LIN {X 0,Y 400.522,Z 455.027,A -85,B 0,C 180,E1 -11218.493,E2 -11218.493} C_VEL
LIN {X 0,Y 403.517,Z 467.527,A -85,B 0,C 180,E1 -11221.017,E2 -11221.017} C_VEL
LIN {X 0,Y 404.106,Z 470.938,A -85,B 0,C 180,E1 -11221.645,E2 -11221.645} C_VEL
LIN {X 0,Y 410.499,Z 503.1,A -85,B 0,C 180,E1 -11222.736,E2 -11222.736} C_VEL
LIN {X 0,Y 411.212,Z 507.909,A -85,B 0,C 180,E1 -11222.879,E2 -11222.879} C_VEL
LIN {X 0,Y 408.574,Z 636.598,A -85,B 0,C 180,E1 -11225.21,E2 -11225.21} C_VEL
LIN {X 0,Y 407.815,Z 651.974,A -85,B 0,C 180,E1 -11225.667,E2 -11225.667} C_VEL
LIN {X 0,Y 406.809,Z 666.551,A -85,B 0,C 180,E1 -11226.294,E2 -11226.294} C_VEL
LIN {X 0,Y 405.685,Z 680.018,A -85,B 0,C 180,E1 -11227.059,E2 -11227.059} C_VEL
LIN {X 0,Y 404.338,Z 693.937,A -85,B 0,C 180,E1 -11228.056,E2 -11228.056} C_VEL
LIN {X 0,Y 402.996,Z 706.696,A -85,B 0,C 180,E1 -11229.186,E2 -11229.186} C_VEL
LIN {X 0,Y 401.616,Z 718.524,A -85,B 0,C 180,E1 -11230.447,E2 -11230.447} C_VEL
LIN {X 0,Y 400.428,Z 729.512,A -85,B 0,C 180,E1 -11231.848,E2 -11231.848} C_VEL
LIN {X 0,Y 399.157,Z 739.653,A -85,B 0,C 180,E1 -11233.374,E2 -11233.374} C_VEL
LIN {X 0,Y 398.037,Z 749.558,A -85,B 0,C 180,E1 -11235.165,E2 -11235.165} C_VEL
LIN {X 0,Y 397.145,Z 757.542,A -85,B 0,C 180,E1 -11236.895,E2 -11236.895} C_VEL
LIN {X 0,Y 396.639,Z 764.626,A -85,B 0,C 180,E1 -11238.76,E2 -11238.76} C_VEL
LIN {X 0,Y 396.122,Z 770.933,A -85,B 0,C 180,E1 -11240.811,E2 -11240.811} C_VEL
LIN {X 0,Y 395.906,Z 775.816,A -85,B 0,C 180,E1 -11242.861,E2 -11242.861} C_VEL
LIN {X 0,Y 395.772,Z 779.396,A -85,B 0,C 180,E1 -11244.906,E2 -11244.906} C_VEL
LIN {X 0,Y 395.703,Z 781.754,A -85,B 0,C 180,E1 -11246.945,E2 -11246.945} C_VEL
LIN {X 0,Y 395.787,Z 782.95,A -85,B 0,C 180,E1 -11248.982,E2 -11248.982} C_VEL
LIN {X 0,Y 395.787,Z 782.947,A -85,B 0,C 180,E1 -11251.017,E2 -11251.017} C_VEL
LIN {X 0,Y 395.711,Z 781.775,A -85,B 0,C 180,E1 -11253.054,E2 -11253.054} C_VEL
LIN {X 0,Y 395.773,Z 779.445,A -85,B 0,C 180,E1 -11255.093,E2 -11255.093} C_VEL
LIN {X 0,Y 395.909,Z 775.906,A -85,B 0,C 180,E1 -11257.137,E2 -11257.137} C_VEL
LIN {X 0,Y 396.129,Z 771.072,A -85,B 0,C 180,E1 -11259.187,E2 -11259.187} C_VEL
LIN {X 0,Y 396.639,Z 764.818,A -85,B 0,C 180,E1 -11261.239,E2 -11261.239} C_VEL
LIN {X 0,Y 397.225,Z 756.862,A -85,B 0,C 180,E1 -11263.32,E2 -11263.32} C_VEL
LIN {X 0,Y 398.204,Z 748.625,A -85,B 0,C 180,E1 -11265.089,E2 -11265.089} C_VEL
LIN {X 0,Y 399.347,Z 738.586,A -85,B 0,C 180,E1 -11266.88,E2 -11266.88} C_VEL
LIN {X 0,Y 400.687,Z 728.32,A -85,B 0,C 180,E1 -11268.403,E2 -11268.403} C_VEL
LIN {X 0,Y 402.04,Z 716.109,A -85,B 0,C 180,E1 -11269.929,E2 -11269.929} C_VEL
LIN {X 0,Y 403.514,Z 703.872,A -85,B 0,C 180,E1 -11271.186,E2 -11271.186} C_VEL
LIN {X 0,Y 404.94,Z 690.58,A -85,B 0,C 180,E1 -11272.311,E2 -11272.311} C_VEL
LIN {X 0,Y 406.337,Z 675.957,A -85,B 0,C 180,E1 -11273.305,E2 -11273.305} C_VEL
LIN {X 0,Y 407.511,Z 661.233,A -85,B 0,C 180,E1 -11274.078,E2 -11274.078} C_VEL
LIN {X 0,Y 408.451,Z 646.947,A -85,B 0,C 180,E1 -11274.627,E2 -11274.627} C_VEL
LIN {X 0,Y 409.13,Z 631.582,A -85,B 0,C 180,E1 -11275.024,E2 -11275.024} C_VEL
LIN {X 0,Y 411.732,Z 507.187,A -85,B 0,C 180,E1 -11277.28,E2 -11277.28} C_VEL
LIN {X 0,Y 407.046,Z 482.434,A -85,B 0,C 180,E1 -11278.129,E2 -11278.129} C_VEL
LIN {X 0,Y 404.35,Z 470.73,A -85,B 0,C 180,E1 -11278.579,E2 -11278.579} C_VEL
LIN {X 0,Y 404.114,Z 469.816,A -85,B 0,C 180,E1 -11278.668,E2 -11278.668} C_VEL
LIN {X 0,Y 400.984,Z 456.078,A -85,B 0,C 180,E1 -11281.486,E2 -11281.486} C_VEL
LIN {X 0,Y 397.135,Z 441.642,A -85,B 0,C 180,E1 -11284.684,E2 -11284.684} C_VEL
LIN {X 0,Y 397.106,Z 441.644,A -85,B 0,C 180,E1 -11288.273,E2 -11288.273} C_VEL
LIN {X 0,Y 397.151,Z 441.64,A -85,B 0,C 180,E1 -11291.993,E2 -11291.993} C_VEL
LIN {X 0,Y 397.105,Z 441.646,A -85,B 0,C 180,E1 -11295.065,E2 -11295.065} C_VEL
LIN {X 0,Y 397.061,Z 441.649,A -85,B 0,C 180,E1 -11298.02,E2 -11298.02} C_VEL
LIN {X 0,Y 397.127,Z 441.641,A -85,B 0,C 180,E1 -11301.137,E2 -11301.137} C_VEL
LIN {X 0,Y 397.114,Z 441.643,A -85,B 0,C 180,E1 -11304.496,E2 -11304.496} C_VEL
LIN {X 0,Y 397.071,Z 441.647,A -85,B 0,C 180,E1 -11307.928,E2 -11307.928} C_VEL
LIN {X 0,Y 397.115,Z 441.642,A -85,B 0,C 180,E1 -11311.456,E2 -11311.456} C_VEL
LIN {X 0,Y 397.146,Z 441.642,A -85,B 0,C 180,E1 -11314.487,E2 -11314.487} C_VEL
LIN {X 0,Y 397.102,Z 441.643,A -85,B 0,C 180,E1 -11317.085,E2 -11317.085} C_VEL
LIN {X 0,Y 397.141,Z 441.638,A -85,B 0,C 180,E1 -11320.353,E2 -11320.353} C_VEL
LIN {X 0,Y 397.159,Z 441.63,A -85,B 0,C 180,E1 -11323.553,E2 -11323.553} C_VEL
LIN {X 0,Y 397.221,Z 441.625,A -85,B 0,C 180,E1 -11326.703,E2 -11326.703} C_VEL
LIN {X 0,Y 397.221,Z 441.628,A -85,B 0,C 180,E1 -11329.809,E2 -11329.809} C_VEL
LIN {X 0,Y 397.356,Z 441.611,A -85,B 0,C 180,E1 -11332.888,E2 -11332.888} C_VEL
LIN {X 0,Y 397.249,Z 441.625,A -85,B 0,C 180,E1 -11334.925,E2 -11334.925} C_VEL
LIN {X 0,Y 397.445,Z 441.597,A -85,B 0,C 180,E1 -11337.974,E2 -11337.974} C_VEL
LIN {X 0,Y 397.573,Z 441.587,A -85,B 0,C 180,E1 -11340,E2 -11340} C_VEL
LIN {X 0,Y 397.376,Z 441.61,A -85,B 0,C 180,E1 -11343.042,E2 -11343.042} C_VEL
LIN {X 0,Y 397.357,Z 441.61,A -85,B 0,C 180,E1 -11347.112,E2 -11347.112} C_VEL
LIN {X 0,Y 397.211,Z 441.633,A -85,B 0,C 180,E1 -11350.191,E2 -11350.191} C_VEL
LIN {X 0,Y 397.22,Z 441.627,A -85,B 0,C 180,E1 -11353.322,E2 -11353.322} C_VEL
LIN {X 0,Y 397.165,Z 441.636,A -85,B 0,C 180,E1 -11356.447,E2 -11356.447} C_VEL
LIN {X 0,Y 397.142,Z 441.638,A -85,B 0,C 180,E1 -11359.648,E2 -11359.648} C_VEL
LIN {X 0,Y 397.129,Z 441.643,A -85,B 0,C 180,E1 -11363.041,E2 -11363.041} C_VEL
LIN {X 0,Y 397.13,Z 441.638,A -85,B 0,C 180,E1 -11366.259,E2 -11366.259} C_VEL
LIN {X 0,Y 397.122,Z 441.647,A -85,B 0,C 180,E1 -11368.544,E2 -11368.544} C_VEL
LIN {X 0,Y 397.106,Z 441.643,A -85,B 0,C 180,E1 -11372.069,E2 -11372.069} C_VEL
LIN {X 0,Y 397.116,Z 441.644,A -85,B 0,C 180,E1 -11375.504,E2 -11375.504} C_VEL
LIN {X 0,Y 397.106,Z 441.683,A -85,B 0,C 180,E1 -11376.836,E2 -11376.836} C_VEL
LIN {X 0,Y 399.634,Z 451.105,A -85,B 0,C 180,E1 -11379.085,E2 -11379.085} C_VEL
LIN {X 0,Y 409.803,Z 473.464,A -85,B 0,C 180,E1 -11380.36,E2 -11380.36} C_VEL
LIN {X 0,Y 411.701,Z 478.608,A -85,B 0,C 180,E1 -11380.608,E2 -11380.608} C_VEL
LIN {X 0,Y 412.192,Z 481.503,A -85,B 0,C 180,E1 -11380.702,E2 -11380.702} C_VEL
LIN {X 0,Y 409.232,Z 616.098,A -85,B 0,C 180,E1 -11383.163,E2 -11383.163} C_VEL
LIN {X 0,Y 408.484,Z 631.664,A -85,B 0,C 180,E1 -11383.649,E2 -11383.649} C_VEL
LIN {X 0,Y 407.56,Z 646.265,A -85,B 0,C 180,E1 -11384.307,E2 -11384.307} C_VEL
LIN {X 0,Y 406.43,Z 660.463,A -85,B 0,C 180,E1 -11385.152,E2 -11385.152} C_VEL
LIN {X 0,Y 405.072,Z 674.297,A -85,B 0,C 180,E1 -11386.191,E2 -11386.191} C_VEL
LIN {X 0,Y 403.678,Z 687.365,A -85,B 0,C 180,E1 -11387.406,E2 -11387.406} C_VEL
LIN {X 0,Y 402.209,Z 699.729,A -85,B 0,C 180,E1 -11388.803,E2 -11388.803} C_VEL
LIN {X 0,Y 400.807,Z 711.212,A -85,B 0,C 180,E1 -11390.372,E2 -11390.372} C_VEL
LIN {X 0,Y 399.332,Z 722.47,A -85,B 0,C 180,E1 -11392.241,E2 -11392.241} C_VEL
LIN {X 0,Y 398.231,Z 731.531,A -85,B 0,C 180,E1 -11394.072,E2 -11394.072} C_VEL
LIN {X 0,Y 397.414,Z 739.183,A -85,B 0,C 180,E1 -11395.948,E2 -11395.948} C_VEL
LIN {X 0,Y 396.693,Z 745.645,A -85,B 0,C 180,E1 -11397.895,E2 -11397.895} C_VEL
LIN {X 0,Y 396.322,Z 750.277,A -85,B 0,C 180,E1 -11399.644,E2 -11399.644} C_VEL
LIN {X 0,Y 395.961,Z 753.947,A -85,B 0,C 180,E1 -11401.366,E2 -11401.366} C_VEL
LIN {X 0,Y 395.669,Z 757.394,A -85,B 0,C 180,E1 -11403.638,E2 -11403.638} C_VEL
LIN {X 0,Y 395.567,Z 759.374,A -85,B 0,C 180,E1 -11405.882,E2 -11405.882} C_VEL
LIN {X 0,Y 395.529,Z 759.982,A -85,B 0,C 180,E1 -11408.091,E2 -11408.091} C_VEL
LIN {X 0,Y 395.617,Z 759.246,A -85,B 0,C 180,E1 -11410.311,E2 -11410.311} C_VEL
LIN {X 0,Y 395.732,Z 757.267,A -85,B 0,C 180,E1 -11412.428,E2 -11412.428} C_VEL
LIN {X 0,Y 396.009,Z 753.977,A -85,B 0,C 180,E1 -11414.562,E2 -11414.562} C_VEL
LIN {X 0,Y 396.334,Z 749.387,A -85,B 0,C 180,E1 -11416.673,E2 -11416.673} C_VEL
LIN {X 0,Y 396.851,Z 743.403,A -85,B 0,C 180,E1 -11418.767,E2 -11418.767} C_VEL
LIN {X 0,Y 397.627,Z 735.873,A -85,B 0,C 180,E1 -11420.848,E2 -11420.848} C_VEL
LIN {X 0,Y 398.535,Z 727.813,A -85,B 0,C 180,E1 -11422.655,E2 -11422.655} C_VEL
LIN {X 0,Y 399.642,Z 718.174,A -85,B 0,C 180,E1 -11424.45,E2 -11424.45} C_VEL
LIN {X 0,Y 400.52,Z 711.345,A -85,B 0,C 180,E1 -11425.54,E2 -11425.54} C_VEL
LIN {X 0,Y 400.336,Z 707.332,A -85,B 0,C 180,E1 -11426.156,E2 -11426.156} C_VEL
LIN {X 0,Y 396.739,Z 695.217,A -85,B 0,C 180,E1 -11427.968,E2 -11427.968} C_VEL
LIN {X 0,Y 396.305,Z 690.74,A -85,B 0,C 180,E1 -11428.526,E2 -11428.526} C_VEL
LIN {X 0,Y 396.421,Z 689.164,A -85,B 0,C 180,E1 -11428.701,E2 -11428.701} C_VEL
LIN {X 0,Y 397.791,Z 677.105,A -85,B 0,C 180,E1 -11429.874,E2 -11429.874} C_VEL
LIN {X 0,Y 399.06,Z 664.569,A -85,B 0,C 180,E1 -11430.884,E2 -11430.884} C_VEL
LIN {X 0,Y 400.329,Z 649.959,A -85,B 0,C 180,E1 -11431.824,E2 -11431.824} C_VEL
LIN {X 0,Y 401.367,Z 635.08,A -85,B 0,C 180,E1 -11432.554,E2 -11432.554} C_VEL
LIN {X 0,Y 402.075,Z 620.623,A -85,B 0,C 180,E1 -11433.069,E2 -11433.069} C_VEL
LIN {X 0,Y 402.585,Z 604.216,A -85,B 0,C 180,E1 -11433.441,E2 -11433.441} C_VEL
LIN {X 0,Y 405.243,Z 482.141,A -85,B 0,C 180,E1 -11435.663,E2 -11435.663} C_VEL
LIN {X 0,Y 404.263,Z 477.972,A -85,B 0,C 180,E1 -11435.817,E2 -11435.817} C_VEL
LIN {X 0,Y 393.374,Z 453.106,A -85,B 0,C 180,E1 -11437.145,E2 -11437.145} C_VEL
LIN {X 0,Y 392.162,Z 450.276,A -85,B 0,C 180,E1 -11437.337,E2 -11437.337} C_VEL
LIN {X 0,Y 390.228,Z 442.507,A -85,B 0,C 180,E1 -11439.185,E2 -11439.185} C_VEL
LIN {X 0,Y 390.182,Z 442.509,A -85,B 0,C 180,E1 -11442.483,E2 -11442.483} C_VEL
LIN {X 0,Y 390.144,Z 442.51,A -85,B 0,C 180,E1 -11445.677,E2 -11445.677} C_VEL
LIN {X 0,Y 390.121,Z 442.513,A -85,B 0,C 180,E1 -11448.922,E2 -11448.922} C_VEL
LIN {X 0,Y 390.045,Z 442.526,A -85,B 0,C 180,E1 -11452.234,E2 -11452.234} C_VEL
LIN {X 0,Y 390.123,Z 442.516,A -85,B 0,C 180,E1 -11455.744,E2 -11455.744} C_VEL
LIN {X 0,Y 390.067,Z 442.516,A -85,B 0,C 180,E1 -11459.109,E2 -11459.109} C_VEL
LIN {X 0,Y 390.047,Z 442.512,A -85,B 0,C 180,E1 -11462.721,E2 -11462.721} C_VEL
LIN {X 0,Y 390.06,Z 442.522,A -85,B 0,C 180,E1 -11465.825,E2 -11465.825} C_VEL
LIN {X 0,Y 390.075,Z 442.512,A -85,B 0,C 180,E1 -11469.219,E2 -11469.219} C_VEL
LIN {X 0,Y 390.053,Z 442.516,A -85,B 0,C 180,E1 -11472.375,E2 -11472.375} C_VEL
LIN {X 0,Y 390.048,Z 442.523,A -85,B 0,C 180,E1 -11475.354,E2 -11475.354} C_VEL
LIN {X 0,Y 390.07,Z 442.511,A -85,B 0,C 180,E1 -11478.191,E2 -11478.191} C_VEL
LIN {X 0,Y 390.097,Z 442.515,A -85,B 0,C 180,E1 -11480.908,E2 -11480.908} C_VEL
LIN {X 0,Y 390.088,Z 442.509,A -85,B 0,C 180,E1 -11484.793,E2 -11484.793} C_VEL
LIN {X 0,Y 390.033,Z 442.524,A -85,B 0,C 180,E1 -11487.875,E2 -11487.875} C_VEL
LIN {X 0,Y 390.059,Z 442.511,A -85,B 0,C 180,E1 -11490.89,E2 -11490.89} C_VEL
LIN {X 0,Y 390.12,Z 442.511,A -85,B 0,C 180,E1 -11494.256,E2 -11494.256} C_VEL
LIN {X 0,Y 390.038,Z 442.517,A -85,B 0,C 180,E1 -11497.765,E2 -11497.765} C_VEL
LIN {X 0,Y 390.106,Z 442.514,A -85,B 0,C 180,E1 -11501.078,E2 -11501.078} C_VEL
LIN {X 0,Y 390.14,Z 442.504,A -85,B 0,C 180,E1 -11504.323,E2 -11504.323} C_VEL
LIN {X 0,Y 390.171,Z 442.51,A -85,B 0,C 180,E1 -11507.517,E2 -11507.517} C_VEL
LIN {X 0,Y 390.315,Z 442.483,A -85,B 0,C 180,E1 -11511.718,E2 -11511.718} C_VEL
LIN {X 0,Y 390.33,Z 442.49,A -85,B 0,C 180,E1 -11513.798,E2 -11513.798} C_VEL
LIN {X 0,Y 390.418,Z 442.469,A -85,B 0,C 180,E1 -11517.937,E2 -11517.937} C_VEL
LIN {X 0,Y 390.55,Z 442.462,A -85,B 0,C 180,E1 -11520,E2 -11520} C_VEL
LIN {X 0,Y 390.315,Z 442.483,A -85,B 0,C 180,E1 -11523.096,E2 -11523.096} C_VEL
LIN {X 0,Y 390.33,Z 442.484,A -85,B 0,C 180,E1 -11526.202,E2 -11526.202} C_VEL
LIN {X 0,Y 390.315,Z 442.489,A -85,B 0,C 180,E1 -11528.282,E2 -11528.282} C_VEL
LIN {X 0,Y 390.17,Z 442.495,A -85,B 0,C 180,E1 -11532.483,E2 -11532.483} C_VEL
LIN {X 0,Y 390.139,Z 442.515,A -85,B 0,C 180,E1 -11535.677,E2 -11535.677} C_VEL
LIN {X 0,Y 390.105,Z 442.501,A -85,B 0,C 180,E1 -11538.922,E2 -11538.922} C_VEL
LIN {X 0,Y 390.039,Z 442.522,A -85,B 0,C 180,E1 -11542.234,E2 -11542.234} C_VEL
LIN {X 0,Y 390.119,Z 442.515,A -85,B 0,C 180,E1 -11545.743,E2 -11545.743} C_VEL
LIN {X 0,Y 390.063,Z 442.519,A -85,B 0,C 180,E1 -11549.109,E2 -11549.109} C_VEL
LIN {X 0,Y 390.043,Z 442.522,A -85,B 0,C 180,E1 -11552.721,E2 -11552.721} C_VEL
LIN {X 0,Y 390.057,Z 442.522,A -85,B 0,C 180,E1 -11555.825,E2 -11555.825} C_VEL
LIN {X 0,Y 390.072,Z 442.52,A -85,B 0,C 180,E1 -11559.219,E2 -11559.219} C_VEL
LIN {X 0,Y 390.043,Z 442.523,A -85,B 0,C 180,E1 -11562.374,E2 -11562.374} C_VEL
LIN {X 0,Y 390.102,Z 442.517,A -85,B 0,C 180,E1 -11566.106,E2 -11566.106} C_VEL
LIN {X 0,Y 390.077,Z 442.522,A -85,B 0,C 180,E1 -11569.175,E2 -11569.175} C_VEL
LIN {X 0,Y 390.043,Z 442.524,A -85,B 0,C 180,E1 -11572.449,E2 -11572.449} C_VEL
LIN {X 0,Y 390.097,Z 442.591,A -85,B 0,C 180,E1 -11575.206,E2 -11575.206} C_VEL
LIN {X 0,Y 393.658,Z 456.492,A -85,B 0,C 180,E1 -11578.22,E2 -11578.22} C_VEL
LIN {X 0,Y 396.682,Z 469.234,A -85,B 0,C 180,E1 -11580.841,E2 -11580.841} C_VEL
LIN {X 0,Y 396.963,Z 470.502,A -85,B 0,C 180,E1 -11581.095,E2 -11581.095} C_VEL
LIN {X 0,Y 398.486,Z 475.203,A -85,B 0,C 180,E1 -11581.316,E2 -11581.316} C_VEL
LIN {X 0,Y 404.772,Z 507.647,A -85,B 0,C 180,E1 -11582.425,E2 -11582.425} C_VEL
LIN {X 0,Y 402.192,Z 632.723,A -85,B 0,C 180,E1 -11584.721,E2 -11584.721} C_VEL
LIN {X 0,Y 401.485,Z 648.689,A -85,B 0,C 180,E1 -11585.158,E2 -11585.158} C_VEL
LIN {X 0,Y 400.542,Z 662.327,A -85,B 0,C 180,E1 -11585.703,E2 -11585.703} C_VEL
LIN {X 0,Y 399.476,Z 675.593,A -85,B 0,C 180,E1 -11586.406,E2 -11586.406} C_VEL
LIN {X 0,Y 398.039,Z 690.371,A -85,B 0,C 180,E1 -11587.416,E2 -11587.416} C_VEL
LIN {X 0,Y 396.587,Z 703.744,A -85,B 0,C 180,E1 -11588.561,E2 -11588.561} C_VEL
LIN {X 0,Y 395.014,Z 717.12,A -85,B 0,C 180,E1 -11589.971,E2 -11589.971} C_VEL
LIN {X 0,Y 393.589,Z 729.204,A -85,B 0,C 180,E1 -11591.521,E2 -11591.521} C_VEL
LIN {X 0,Y 392.296,Z 739.364,A -85,B 0,C 180,E1 -11593.075,E2 -11593.075} C_VEL
LIN {X 0,Y 391.114,Z 749.284,A -85,B 0,C 180,E1 -11594.897,E2 -11594.897} C_VEL
LIN {X 0,Y 390.215,Z 756.811,A -85,B 0,C 180,E1 -11596.549,E2 -11596.549} C_VEL
LIN {X 0,Y 389.609,Z 764.374,A -85,B 0,C 180,E1 -11598.555,E2 -11598.555} C_VEL
LIN {X 0,Y 389.054,Z 770.693,A -85,B 0,C 180,E1 -11600.643,E2 -11600.643} C_VEL
LIN {X 0,Y 388.825,Z 775.587,A -85,B 0,C 180,E1 -11602.731,E2 -11602.731} C_VEL
LIN {X 0,Y 388.676,Z 779.175,A -85,B 0,C 180,E1 -11604.812,E2 -11604.812} C_VEL
LIN {X 0,Y 388.61,Z 781.54,A -85,B 0,C 180,E1 -11606.889,E2 -11606.889} C_VEL
LIN {X 0,Y 388.699,Z 782.741,A -85,B 0,C 180,E1 -11608.963,E2 -11608.963} C_VEL
LIN {X 0,Y 388.699,Z 782.741,A -85,B 0,C 180,E1 -11611.035,E2 -11611.035} C_VEL
LIN {X 0,Y 388.618,Z 781.573,A -85,B 0,C 180,E1 -11613.109,E2 -11613.109} C_VEL
LIN {X 0,Y 388.677,Z 779.248,A -85,B 0,C 180,E1 -11615.187,E2 -11615.187} C_VEL
LIN {X 0,Y 388.827,Z 775.716,A -85,B 0,C 180,E1 -11617.268,E2 -11617.268} C_VEL
LIN {X 0,Y 389.06,Z 770.887,A -85,B 0,C 180,E1 -11619.356,E2 -11619.356} C_VEL
LIN {X 0,Y 389.613,Z 764.639,A -85,B 0,C 180,E1 -11621.444,E2 -11621.444} C_VEL
LIN {X 0,Y 390.268,Z 756.792,A -85,B 0,C 180,E1 -11623.538,E2 -11623.538} C_VEL
LIN {X 0,Y 391.286,Z 748.457,A -85,B 0,C 180,E1 -11625.362,E2 -11625.362} C_VEL
LIN {X 0,Y 392.488,Z 738.425,A -85,B 0,C 180,E1 -11627.184,E2 -11627.184} C_VEL
LIN {X 0,Y 393.979,Z 727.182,A -85,B 0,C 180,E1 -11628.872,E2 -11628.872} C_VEL
LIN {X 0,Y 395.456,Z 714.852,A -85,B 0,C 180,E1 -11630.411,E2 -11630.411} C_VEL
LIN {X 0,Y 396.988,Z 702.459,A -85,B 0,C 180,E1 -11631.687,E2 -11631.687} C_VEL
LIN {X 0,Y 398.514,Z 688.923,A -85,B 0,C 180,E1 -11632.828,E2 -11632.828} C_VEL
LIN {X 0,Y 399.904,Z 674.945,A -85,B 0,C 180,E1 -11633.772,E2 -11633.772} C_VEL
LIN {X 0,Y 401.084,Z 660.449,A -85,B 0,C 180,E1 -11634.533,E2 -11634.533} C_VEL
LIN {X 0,Y 402.134,Z 645.278,A -85,B 0,C 180,E1 -11635.109,E2 -11635.109} C_VEL
LIN {X 0,Y 402.793,Z 628.997,A -85,B 0,C 180,E1 -11635.514,E2 -11635.514} C_VEL
LIN {X 0,Y 405.441,Z 508.807,A -85,B 0,C 180,E1 -11637.72,E2 -11637.72} C_VEL
LIN {X 0,Y 401.384,Z 486.309,A -85,B 0,C 180,E1 -11638.497,E2 -11638.497} C_VEL
LIN {X 0,Y 398.475,Z 473.46,A -85,B 0,C 180,E1 -11639,E2 -11639} C_VEL
LIN {X 0,Y 396.956,Z 469.79,A -85,B 0,C 180,E1 -11639.221,E2 -11639.221} C_VEL
LIN {X 0,Y 394.202,Z 457.847,A -85,B 0,C 180,E1 -11641.73,E2 -11641.73} C_VEL
LIN {X 0,Y 390.109,Z 442.514,A -85,B 0,C 180,E1 -11645.203,E2 -11645.203} C_VEL
LIN {X 0,Y 390.07,Z 442.521,A -85,B 0,C 180,E1 -11649.219,E2 -11649.219} C_VEL
LIN {X 0,Y 390.115,Z 442.511,A -85,B 0,C 180,E1 -11652.386,E2 -11652.386} C_VEL
LIN {X 0,Y 390.055,Z 442.524,A -85,B 0,C 180,E1 -11655.356,E2 -11655.356} C_VEL
LIN {X 0,Y 390.025,Z 442.528,A -85,B 0,C 180,E1 -11658.186,E2 -11658.186} C_VEL
LIN {X 0,Y 390.086,Z 442.519,A -85,B 0,C 180,E1 -11660.907,E2 -11660.907} C_VEL
LIN {X 0,Y 390.079,Z 442.519,A -85,B 0,C 180,E1 -11664.793,E2 -11664.793} C_VEL
LIN {X 0,Y 390.025,Z 442.524,A -85,B 0,C 180,E1 -11667.875,E2 -11667.875} C_VEL
LIN {X 0,Y 390.051,Z 442.523,A -85,B 0,C 180,E1 -11670.89,E2 -11670.89} C_VEL
LIN {X 0,Y 390.112,Z 442.517,A -85,B 0,C 180,E1 -11674.256,E2 -11674.256} C_VEL
LIN {X 0,Y 390.032,Z 442.525,A -85,B 0,C 180,E1 -11677.766,E2 -11677.766} C_VEL
LIN {X 0,Y 390.098,Z 442.516,A -85,B 0,C 180,E1 -11681.078,E2 -11681.078} C_VEL
LIN {X 0,Y 390.132,Z 442.512,A -85,B 0,C 180,E1 -11684.323,E2 -11684.323} C_VEL
LIN {X 0,Y 390.17,Z 442.503,A -85,B 0,C 180,E1 -11687.517,E2 -11687.517} C_VEL
LIN {X 0,Y 390.308,Z 442.489,A -85,B 0,C 180,E1 -11691.718,E2 -11691.718} C_VEL
LIN {X 0,Y 390.323,Z 442.486,A -85,B 0,C 180,E1 -11693.798,E2 -11693.798} C_VEL
LIN {X 0,Y 390.414,Z 442.473,A -85,B 0,C 180,E1 -11697.937,E2 -11697.937} C_VEL
LIN {X 0,Y 390.543,Z 442.463,A -85,B 0,C 180,E1 -11700,E2 -11700} C_VEL
LIN {X 0,Y 390.31,Z 442.49,A -85,B 0,C 180,E1 -11703.097,E2 -11703.097} C_VEL
LIN {X 0,Y 390.303,Z 442.489,A -85,B 0,C 180,E1 -11706.619,E2 -11706.619} C_VEL
LIN {X 0,Y 390.198,Z 442.504,A -85,B 0,C 180,E1 -11709.329,E2 -11709.329} C_VEL
LIN {X 0,Y 390.188,Z 442.503,A -85,B 0,C 180,E1 -11713.439,E2 -11713.439} C_VEL
LIN {X 0,Y 390.144,Z 442.51,A -85,B 0,C 180,E1 -11717.309,E2 -11717.309} C_VEL
LIN {X 0,Y 390.086,Z 442.523,A -85,B 0,C 180,E1 -11720.473,E2 -11720.473} C_VEL
LIN {X 0,Y 390.084,Z 442.52,A -85,B 0,C 180,E1 -11723.352,E2 -11723.352} C_VEL
LIN {X 0,Y 390.108,Z 442.511,A -85,B 0,C 180,E1 -11726.769,E2 -11726.769} C_VEL
LIN {X 0,Y 390.04,Z 442.521,A -85,B 0,C 180,E1 -11730.3,E2 -11730.3} C_VEL
LIN {X 0,Y 390.08,Z 442.523,A -85,B 0,C 180,E1 -11733.954,E2 -11733.954} C_VEL
LIN {X 0,Y 390.062,Z 442.637,A -85,B 0,C 180,E1 -11736.329,E2 -11736.329} C_VEL
LIN {X 0,Y 392.357,Z 451.225,A -85,B 0,C 180,E1 -11738.463,E2 -11738.463} C_VEL
LIN {X 0,Y 401.061,Z 469.691,A -85,B 0,C 180,E1 -11739.59,E2 -11739.59} C_VEL
LIN {X 0,Y 405.727,Z 481.092,A -85,B 0,C 180,E1 -11740.197,E2 -11740.197} C_VEL
LIN {X 0,Y 405.873,Z 485.028,A -85,B 0,C 180,E1 -11740.288,E2 -11740.288} C_VEL
LIN {X 0,Y 402.848,Z 616.252,A -85,B 0,C 180,E1 -11742.725,E2 -11742.725} C_VEL
LIN {X 0,Y 402.061,Z 631.983,A -85,B 0,C 180,E1 -11743.224,E2 -11743.224} C_VEL
LIN {X 0,Y 401.086,Z 646.661,A -85,B 0,C 180,E1 -11743.897,E2 -11743.897} C_VEL
LIN {X 0,Y 399.888,Z 660.995,A -85,B 0,C 180,E1 -11744.766,E2 -11744.766} C_VEL
LIN {X 0,Y 398.452,Z 674.977,A -85,B 0,C 180,E1 -11745.838,E2 -11745.838} C_VEL
LIN {X 0,Y 397.047,Z 687.667,A -85,B 0,C 180,E1 -11747.042,E2 -11747.042} C_VEL
LIN {X 0,Y 395.526,Z 699.722,A -85,B 0,C 180,E1 -11748.425,E2 -11748.425} C_VEL
LIN {X 0,Y 393.998,Z 711.685,A -85,B 0,C 180,E1 -11750.087,E2 -11750.087} C_VEL
LIN {X 0,Y 392.676,Z 721.198,A -85,B 0,C 180,E1 -11751.674,E2 -11751.674} C_VEL
LIN {X 0,Y 391.59,Z 729.701,A -85,B 0,C 180,E1 -11753.364,E2 -11753.364} C_VEL
LIN {X 0,Y 390.628,Z 737.237,A -85,B 0,C 180,E1 -11755.149,E2 -11755.149} C_VEL
LIN {X 0,Y 390.029,Z 742.654,A -85,B 0,C 180,E1 -11756.663,E2 -11756.663} C_VEL
LIN {X 0,Y 389.482,Z 747.911,A -85,B 0,C 180,E1 -11758.448,E2 -11758.448} C_VEL
LIN {X 0,Y 389.144,Z 751.909,A -85,B 0,C 180,E1 -11760.1,E2 -11760.1} C_VEL
LIN {X 0,Y 388.723,Z 756.031,A -85,B 0,C 180,E1 -11762.364,E2 -11762.364} C_VEL
LIN {X 0,Y 388.545,Z 758.807,A -85,B 0,C 180,E1 -11764.743,E2 -11764.743} C_VEL
LIN {X 0,Y 388.459,Z 760.106,A -85,B 0,C 180,E1 -11767.324,E2 -11767.324} C_VEL
LIN {X 0,Y 388.424,Z 760.077,A -85,B 0,C 180,E1 -11768.786,E2 -11768.786} C_VEL
LIN {X 0,Y 388.557,Z 758.946,A -85,B 0,C 180,E1 -11771,E2 -11771} C_VEL
LIN {X 0,Y 388.777,Z 756.31,A -85,B 0,C 180,E1 -11773.355,E2 -11773.355} C_VEL
LIN {X 0,Y 389.054,Z 752.857,A -85,B 0,C 180,E1 -11775.352,E2 -11775.352} C_VEL
LIN {X 0,Y 389.423,Z 747.849,A -85,B 0,C 180,E1 -11777.493,E2 -11777.493} C_VEL
LIN {X 0,Y 390.069,Z 741.392,A -85,B 0,C 180,E1 -11779.621,E2 -11779.621} C_VEL
LIN {X 0,Y 390.968,Z 733.318,A -85,B 0,C 180,E1 -11781.732,E2 -11781.732} C_VEL
LIN {X 0,Y 391.978,Z 724.734,A -85,B 0,C 180,E1 -11783.567,E2 -11783.567} C_VEL
LIN {X 0,Y 393.33,Z 714.397,A -85,B 0,C 180,E1 -11785.389,E2 -11785.389} C_VEL
LIN {X 0,Y 394.65,Z 703.852,A -85,B 0,C 180,E1 -11786.938,E2 -11786.938} C_VEL
LIN {X 0,Y 396.017,Z 692.404,A -85,B 0,C 180,E1 -11788.348,E2 -11788.348} C_VEL
LIN {X 0,Y 396.421,Z 689.164,A -85,B 0,C 180,E1 -11788.701,E2 -11788.701} C_VEL
LIN {X 0,Y 396.361,Z 684.491,A -85,B 0,C 180,E1 -11789.225,E2 -11789.225} C_VEL
LIN {X 0,Y 394.527,Z 676.837,A -85,B 0,C 180,E1 -11790.102,E2 -11790.102} C_VEL
LIN {X 0,Y 392.681,Z 668.92,A -85,B 0,C 180,E1 -11790.92,E2 -11790.92} C_VEL
LIN {X 0,Y 392.586,Z 663.748,A -85,B 0,C 180,E1 -11791.344,E2 -11791.344} C_VEL
LIN {X 0,Y 393.769,Z 650.516,A -85,B 0,C 180,E1 -11792.204,E2 -11792.204} C_VEL
LIN {X 0,Y 394.777,Z 636.592,A -85,B 0,C 180,E1 -11792.91,E2 -11792.91} C_VEL
LIN {X 0,Y 395.589,Z 621.413,A -85,B 0,C 180,E1 -11793.47,E2 -11793.47} C_VEL
LIN {X 0,Y 396.115,Z 605.348,A -85,B 0,C 180,E1 -11793.847,E2 -11793.847} C_VEL
LIN {X 0,Y 398.868,Z 482.784,A -85,B 0,C 180,E1 -11796.116,E2 -11796.116} C_VEL
LIN {X 0,Y 397.112,Z 477.867,A -85,B 0,C 180,E1 -11796.347,E2 -11796.347} C_VEL
LIN {X 0,Y 386.692,Z 454.263,A -85,B 0,C 180,E1 -11797.656,E2 -11797.656} C_VEL
LIN {X 0,Y 385.015,Z 450.617,A -85,B 0,C 180,E1 -11797.885,E2 -11797.885} C_VEL
LIN {X 0,Y 383.147,Z 443.38,A -85,B 0,C 180,E1 -11799.669,E2 -11799.669} C_VEL
LIN {X 0,Y 383.13,Z 443.385,A -85,B 0,C 180,E1 -11803.537,E2 -11803.537} C_VEL
LIN {X 0,Y 383.099,Z 443.39,A -85,B 0,C 180,E1 -11807.455,E2 -11807.455} C_VEL
LIN {X 0,Y 383.045,Z 443.393,A -85,B 0,C 180,E1 -11810.652,E2 -11810.652} C_VEL
LIN {X 0,Y 383.037,Z 443.393,A -85,B 0,C 180,E1 -11813.807,E2 -11813.807} C_VEL
LIN {X 0,Y 383.06,Z 443.392,A -85,B 0,C 180,E1 -11817.302,E2 -11817.302} C_VEL
LIN {X 0,Y 382.99,Z 443.402,A -85,B 0,C 180,E1 -11820.918,E2 -11820.918} C_VEL
LIN {X 0,Y 383.021,Z 443.397,A -85,B 0,C 180,E1 -11824.668,E2 -11824.668} C_VEL
LIN {X 0,Y 383.005,Z 443.39,A -85,B 0,C 180,E1 -11827.904,E2 -11827.904} C_VEL
LIN {X 0,Y 383.001,Z 443.403,A -85,B 0,C 180,E1 -11831.345,E2 -11831.345} C_VEL
LIN {X 0,Y 383,Z 443.398,A -85,B 0,C 180,E1 -11834.304,E2 -11834.304} C_VEL
LIN {X 0,Y 383.042,Z 443.396,A -85,B 0,C 180,E1 -11837.244,E2 -11837.244} C_VEL
LIN {X 0,Y 383.024,Z 443.397,A -85,B 0,C 180,E1 -11840.412,E2 -11840.412} C_VEL
LIN {X 0,Y 383.029,Z 443.388,A -85,B 0,C 180,E1 -11844.044,E2 -11844.044} C_VEL
LIN {X 0,Y 383.006,Z 443.403,A -85,B 0,C 180,E1 -11847.573,E2 -11847.573} C_VEL
LIN {X 0,Y 382.993,Z 443.391,A -85,B 0,C 180,E1 -11850.3,E2 -11850.3} C_VEL
LIN {X 0,Y 383.082,Z 443.39,A -85,B 0,C 180,E1 -11854.021,E2 -11854.021} C_VEL
LIN {X 0,Y 382.996,Z 443.388,A -85,B 0,C 180,E1 -11857.334,E2 -11857.334} C_VEL
LIN {X 0,Y 383.061,Z 443.39,A -85,B 0,C 180,E1 -11860.716,E2 -11860.716} C_VEL
LIN {X 0,Y 383.081,Z 443.381,A -85,B 0,C 180,E1 -11864.026,E2 -11864.026} C_VEL
LIN {X 0,Y 383.137,Z 443.384,A -85,B 0,C 180,E1 -11867.284,E2 -11867.284} C_VEL
LIN {X 0,Y 383.152,Z 443.368,A -85,B 0,C 180,E1 -11870.498,E2 -11870.498} C_VEL
LIN {X 0,Y 383.273,Z 443.363,A -85,B 0,C 180,E1 -11872.625,E2 -11872.625} C_VEL
LIN {X 0,Y 383.199,Z 443.373,A -85,B 0,C 180,E1 -11874.738,E2 -11874.738} C_VEL
LIN {X 0,Y 383.385,Z 443.344,A -85,B 0,C 180,E1 -11877.899,E2 -11877.899} C_VEL
LIN {X 0,Y 383.52,Z 443.338,A -85,B 0,C 180,E1 -11880,E2 -11880} C_VEL
LIN {X 0,Y 383.251,Z 443.363,A -85,B 0,C 180,E1 -11883.153,E2 -11883.153} C_VEL
LIN {X 0,Y 383.287,Z 443.36,A -85,B 0,C 180,E1 -11886.316,E2 -11886.316} C_VEL
LIN {X 0,Y 383.26,Z 443.367,A -85,B 0,C 180,E1 -11888.435,E2 -11888.435} C_VEL
LIN {X 0,Y 383.097,Z 443.375,A -85,B 0,C 180,E1 -11891.642,E2 -11891.642} C_VEL
LIN {X 0,Y 383.11,Z 443.385,A -85,B 0,C 180,E1 -11894.881,E2 -11894.881} C_VEL
LIN {X 0,Y 383.063,Z 443.379,A -85,B 0,C 180,E1 -11898.173,E2 -11898.173} C_VEL
LIN {X 0,Y 382.993,Z 443.404,A -85,B 0,C 180,E1 -11901.531,E2 -11901.531} C_VEL
LIN {X 0,Y 383.052,Z 443.393,A -85,B 0,C 180,E1 -11904.96,E2 -11904.96} C_VEL
LIN {X 0,Y 383.049,Z 443.392,A -85,B 0,C 180,E1 -11908.492,E2 -11908.492} C_VEL
LIN {X 0,Y 383.01,Z 443.4,A -85,B 0,C 180,E1 -11912.149,E2 -11912.149} C_VEL
LIN {X 0,Y 383.018,Z 443.397,A -85,B 0,C 180,E1 -11914.668,E2 -11914.668} C_VEL
LIN {X 0,Y 383.002,Z 443.401,A -85,B 0,C 180,E1 -11917.904,E2 -11917.904} C_VEL
LIN {X 0,Y 382.985,Z 443.404,A -85,B 0,C 180,E1 -11921.347,E2 -11921.347} C_VEL
LIN {X 0,Y 383.007,Z 443.4,A -85,B 0,C 180,E1 -11924.305,E2 -11924.305} C_VEL
LIN {X 0,Y 383.075,Z 443.394,A -85,B 0,C 180,E1 -11927.249,E2 -11927.249} C_VEL
LIN {X 0,Y 383.018,Z 443.401,A -85,B 0,C 180,E1 -11930.413,E2 -11930.413} C_VEL
LIN {X 0,Y 383.025,Z 443.398,A -85,B 0,C 180,E1 -11934.044,E2 -11934.044} C_VEL
LIN {X 0,Y 383.054,Z 443.513,A -85,B 0,C 180,E1 -11934.734,E2 -11934.734} C_VEL
LIN {X 0,Y 386.33,Z 456.123,A -85,B 0,C 180,E1 -11937.544,E2 -11937.544} C_VEL
LIN {X 0,Y 389.487,Z 469.233,A -85,B 0,C 180,E1 -11940.314,E2 -11940.314} C_VEL
LIN {X 0,Y 389.713,Z 470.299,A -85,B 0,C 180,E1 -11940.532,E2 -11940.532} C_VEL
LIN {X 0,Y 392.407,Z 477.46,A -85,B 0,C 180,E1 -11940.898,E2 -11940.898} C_VEL
LIN {X 0,Y 398.464,Z 509.25,A -85,B 0,C 180,E1 -11942.005,E2 -11942.005} C_VEL
LIN {X 0,Y 395.615,Z 636.2,A -85,B 0,C 180,E1 -11944.376,E2 -11944.376} C_VEL
LIN {X 0,Y 394.808,Z 651.658,A -85,B 0,C 180,E1 -11944.849,E2 -11944.849} C_VEL
LIN {X 0,Y 393.758,Z 665.967,A -85,B 0,C 180,E1 -11945.482,E2 -11945.482} C_VEL
LIN {X 0,Y 392.513,Z 679.441,A -85,B 0,C 180,E1 -11946.264,E2 -11946.264} C_VEL
LIN {X 0,Y 391.081,Z 693.153,A -85,B 0,C 180,E1 -11947.271,E2 -11947.271} C_VEL
LIN {X 0,Y 389.61,Z 705.987,A -85,B 0,C 180,E1 -11948.436,E2 -11948.436} C_VEL
LIN {X 0,Y 387.986,Z 718.945,A -85,B 0,C 180,E1 -11949.869,E2 -11949.869} C_VEL
LIN {X 0,Y 386.773,Z 728.896,A -85,B 0,C 180,E1 -11951.183,E2 -11951.183} C_VEL
LIN {X 0,Y 385.436,Z 739.075,A -85,B 0,C 180,E1 -11952.764,E2 -11952.764} C_VEL
LIN {X 0,Y 384.175,Z 749.009,A -85,B 0,C 180,E1 -11954.617,E2 -11954.617} C_VEL
LIN {X 0,Y 383.109,Z 757.94,A -85,B 0,C 180,E1 -11956.643,E2 -11956.643} C_VEL
LIN {X 0,Y 382.589,Z 764.119,A -85,B 0,C 180,E1 -11958.342,E2 -11958.342} C_VEL
LIN {X 0,Y 382.003,Z 770.45,A -85,B 0,C 180,E1 -11960.469,E2 -11960.469} C_VEL
LIN {X 0,Y 381.733,Z 775.353,A -85,B 0,C 180,E1 -11962.595,E2 -11962.595} C_VEL
LIN {X 0,Y 381.586,Z 778.951,A -85,B 0,C 180,E1 -11964.716,E2 -11964.716} C_VEL
LIN {X 0,Y 381.522,Z 781.324,A -85,B 0,C 180,E1 -11966.832,E2 -11966.832} C_VEL
LIN {X 0,Y 381.613,Z 782.532,A -85,B 0,C 180,E1 -11968.944,E2 -11968.944} C_VEL
LIN {X 0,Y 381.614,Z 782.535,A -85,B 0,C 180,E1 -11971.055,E2 -11971.055} C_VEL
LIN {X 0,Y 381.529,Z 781.373,A -85,B 0,C 180,E1 -11973.167,E2 -11973.167} C_VEL
LIN {X 0,Y 381.587,Z 779.053,A -85,B 0,C 180,E1 -11975.283,E2 -11975.283} C_VEL
LIN {X 0,Y 381.735,Z 775.526,A -85,B 0,C 180,E1 -11977.404,E2 -11977.404} C_VEL
LIN {X 0,Y 382.007,Z 770.703,A -85,B 0,C 180,E1 -11979.53,E2 -11979.53} C_VEL
LIN {X 0,Y 382.595,Z 764.46,A -85,B 0,C 180,E1 -11981.657,E2 -11981.657} C_VEL
LIN {X 0,Y 383.326,Z 756.619,A -85,B 0,C 180,E1 -11983.788,E2 -11983.788} C_VEL
LIN {X 0,Y 384.381,Z 748.294,A -85,B 0,C 180,E1 -11985.645,E2 -11985.645} C_VEL
LIN {X 0,Y 385.658,Z 738.281,A -85,B 0,C 180,E1 -11987.498,E2 -11987.498} C_VEL
LIN {X 0,Y 387.079,Z 728.038,A -85,B 0,C 180,E1 -11989.075,E2 -11989.075} C_VEL
LIN {X 0,Y 388.605,Z 715.867,A -85,B 0,C 180,E1 -11990.649,E2 -11990.649} C_VEL
LIN {X 0,Y 390.217,Z 703.681,A -85,B 0,C 180,E1 -11991.944,E2 -11991.944} C_VEL
LIN {X 0,Y 391.781,Z 690.457,A -85,B 0,C 180,E1 -11993.103,E2 -11993.103} C_VEL
LIN {X 0,Y 393.143,Z 677.904,A -85,B 0,C 180,E1 -11993.996,E2 -11993.996} C_VEL
LIN {X 0,Y 394.341,Z 664.185,A -85,B 0,C 180,E1 -11994.78,E2 -11994.78} C_VEL
LIN {X 0,Y 395.437,Z 649.982,A -85,B 0,C 180,E1 -11995.388,E2 -11995.388} C_VEL
LIN {X 0,Y 396.207,Z 635.341,A -85,B 0,C 180,E1 -11995.829,E2 -11995.829} C_VEL
LIN {X 0,Y 398.632,Z 533.429,A -85,B 0,C 180,E1 -11997.745,E2 -11997.745} C_VEL
LIN {X 0,Y 399.105,Z 508.593,A -85,B 0,C 180,E1 -11998.22,E2 -11998.22} C_VEL
LIN {X 0,Y 394.581,Z 484.688,A -85,B 0,C 180,E1 -11999.089,E2 -11999.089} C_VEL
LIN {X 0,Y 392.713,Z 476.543,A -85,B 0,C 180,E1 -11999.42,E2 -11999.42} C_VEL
LIN {X 0,Y 389.729,Z 469.591,A -85,B 0,C 180,E1 -11999.835,E2 -11999.835} C_VEL
LIN {X 0,Y 386.907,Z 457.778,A -85,B 0,C 180,E1 -12002.401,E2 -12002.401} C_VEL
LIN {X 0,Y 383.65,Z 445.492,A -85,B 0,C 180,E1 -12005.241,E2 -12005.241} C_VEL
LIN {X 0,Y 383.028,Z 443.397,A -85,B 0,C 180,E1 -12005.792,E2 -12005.792} C_VEL
LIN {X 0,Y 383.018,Z 443.395,A -85,B 0,C 180,E1 -12009.587,E2 -12009.587} C_VEL
LIN {X 0,Y 383.06,Z 443.387,A -85,B 0,C 180,E1 -12012.788,E2 -12012.788} C_VEL
LIN {X 0,Y 383.001,Z 443.398,A -85,B 0,C 180,E1 -12015.79,E2 -12015.79} C_VEL
LIN {X 0,Y 382.983,Z 443.406,A -85,B 0,C 180,E1 -12018.795,E2 -12018.795} C_VEL
LIN {X 0,Y 382.996,Z 443.401,A -85,B 0,C 180,E1 -12022.095,E2 -12022.095} C_VEL
LIN {X 0,Y 383.012,Z 443.399,A -85,B 0,C 180,E1 -12025.332,E2 -12025.332} C_VEL
LIN {X 0,Y 382.976,Z 443.402,A -85,B 0,C 180,E1 -12029.081,E2 -12029.081} C_VEL
LIN {X 0,Y 383.05,Z 443.391,A -85,B 0,C 180,E1 -12032.698,E2 -12032.698} C_VEL
LIN {X 0,Y 383.045,Z 443.394,A -85,B 0,C 180,E1 -12035.039,E2 -12035.039} C_VEL
LIN {X 0,Y 382.986,Z 443.403,A -85,B 0,C 180,E1 -12038.469,E2 -12038.469} C_VEL
LIN {X 0,Y 383.082,Z 443.392,A -85,B 0,C 180,E1 -12041.828,E2 -12041.828} C_VEL
LIN {X 0,Y 383.105,Z 443.387,A -85,B 0,C 180,E1 -12045.118,E2 -12045.118} C_VEL
LIN {X 0,Y 383.1,Z 443.391,A -85,B 0,C 180,E1 -12048.358,E2 -12048.358} C_VEL
LIN {X 0,Y 383.296,Z 443.363,A -85,B 0,C 180,E1 -12051.933,E2 -12051.933} C_VEL
LIN {X 0,Y 383.193,Z 443.375,A -85,B 0,C 180,E1 -12054.739,E2 -12054.739} C_VEL
LIN {X 0,Y 383.381,Z 443.348,A -85,B 0,C 180,E1 -12057.899,E2 -12057.899} C_VEL
LIN {X 0,Y 383.512,Z 443.339,A -85,B 0,C 180,E1 -12060,E2 -12060} C_VEL
LIN {X 0,Y 383.247,Z 443.37,A -85,B 0,C 180,E1 -12063.154,E2 -12063.154} C_VEL
LIN {X 0,Y 383.263,Z 443.368,A -85,B 0,C 180,E1 -12066.613,E2 -12066.613} C_VEL
LIN {X 0,Y 383.253,Z 443.368,A -85,B 0,C 180,E1 -12068.436,E2 -12068.436} C_VEL
LIN {X 0,Y 383.09,Z 443.386,A -85,B 0,C 180,E1 -12071.643,E2 -12071.643} C_VEL
LIN {X 0,Y 383.107,Z 443.389,A -85,B 0,C 180,E1 -12074.882,E2 -12074.882} C_VEL
LIN {X 0,Y 383.083,Z 443.394,A -85,B 0,C 180,E1 -12078.173,E2 -12078.173} C_VEL
LIN {X 0,Y 382.99,Z 443.401,A -85,B 0,C 180,E1 -12081.531,E2 -12081.531} C_VEL
LIN {X 0,Y 383.047,Z 443.399,A -85,B 0,C 180,E1 -12084.961,E2 -12084.961} C_VEL
LIN {X 0,Y 383.044,Z 443.401,A -85,B 0,C 180,E1 -12088.493,E2 -12088.493} C_VEL
LIN {X 0,Y 383.003,Z 443.397,A -85,B 0,C 180,E1 -12092.428,E2 -12092.428} C_VEL
LIN {X 0,Y 383.031,Z 443.548,A -85,B 0,C 180,E1 -12095.793,E2 -12095.793} C_VEL
LIN {X 0,Y 385.222,Z 451.59,A -85,B 0,C 180,E1 -12097.827,E2 -12097.827} C_VEL
LIN {X 0,Y 393.005,Z 467.672,A -85,B 0,C 180,E1 -12098.872,E2 -12098.872} C_VEL
LIN {X 0,Y 399.552,Z 482.795,A -85,B 0,C 180,E1 -12099.738,E2 -12099.738} C_VEL
LIN {X 0,Y 399.481,Z 492.838,A -85,B 0,C 180,E1 -12099.94,E2 -12099.94} C_VEL
LIN {X 0,Y 396.516,Z 616.103,A -85,B 0,C 180,E1 -12102.267,E2 -12102.267} C_VEL
LIN {X 0,Y 395.725,Z 631.695,A -85,B 0,C 180,E1 -12102.762,E2 -12102.762} C_VEL
LIN {X 0,Y 394.702,Z 646.446,A -85,B 0,C 180,E1 -12103.441,E2 -12103.441} C_VEL
LIN {X 0,Y 393.445,Z 660.751,A -85,B 0,C 180,E1 -12104.313,E2 -12104.313} C_VEL
LIN {X 0,Y 391.898,Z 675.295,A -85,B 0,C 180,E1 -12105.443,E2 -12105.443} C_VEL
LIN {X 0,Y 390.408,Z 688.086,A -85,B 0,C 180,E1 -12106.677,E2 -12106.677} C_VEL
LIN {X 0,Y 388.709,Z 700.924,A -85,B 0,C 180,E1 -12108.188,E2 -12108.188} C_VEL
LIN {X 0,Y 387.328,Z 711.239,A -85,B 0,C 180,E1 -12109.649,E2 -12109.649} C_VEL
LIN {X 0,Y 385.819,Z 721.555,A -85,B 0,C 180,E1 -12111.387,E2 -12111.387} C_VEL
LIN {X 0,Y 384.578,Z 730.889,A -85,B 0,C 180,E1 -12113.294,E2 -12113.294} C_VEL
LIN {X 0,Y 383.532,Z 739.268,A -85,B 0,C 180,E1 -12115.386,E2 -12115.386} C_VEL
LIN {X 0,Y 382.625,Z 746.544,A -85,B 0,C 180,E1 -12117.664,E2 -12117.664} C_VEL
LIN {X 0,Y 382.122,Z 751.869,A -85,B 0,C 180,E1 -12119.818,E2 -12119.818} C_VEL
LIN {X 0,Y 381.661,Z 756.058,A -85,B 0,C 180,E1 -12122.115,E2 -12122.115} C_VEL
LIN {X 0,Y 381.467,Z 758.907,A -85,B 0,C 180,E1 -12124.524,E2 -12124.524} C_VEL
LIN {X 0,Y 381.372,Z 760.29,A -85,B 0,C 180,E1 -12127.134,E2 -12127.134} C_VEL
LIN {X 0,Y 381.379,Z 760.068,A -85,B 0,C 180,E1 -12129.506,E2 -12129.506} C_VEL
LIN {X 0,Y 381.488,Z 758.548,A -85,B 0,C 180,E1 -12131.75,E2 -12131.75} C_VEL
LIN {X 0,Y 381.749,Z 755.753,A -85,B 0,C 180,E1 -12133.97,E2 -12133.97} C_VEL
LIN {X 0,Y 382.099,Z 751.66,A -85,B 0,C 180,E1 -12136.167,E2 -12136.167} C_VEL
LIN {X 0,Y 382.603,Z 746.203,A -85,B 0,C 180,E1 -12138.343,E2 -12138.343} C_VEL
LIN {X 0,Y 383.347,Z 739.263,A -85,B 0,C 180,E1 -12140.503,E2 -12140.503} C_VEL
LIN {X 0,Y 384.243,Z 731.794,A -85,B 0,C 180,E1 -12142.38,E2 -12142.38} C_VEL
LIN {X 0,Y 385.403,Z 722.838,A -85,B 0,C 180,E1 -12144.244,E2 -12144.244} C_VEL
LIN {X 0,Y 386.625,Z 713.723,A -85,B 0,C 180,E1 -12145.831,E2 -12145.831} C_VEL
LIN {X 0,Y 388.021,Z 703.005,A -85,B 0,C 180,E1 -12147.405,E2 -12147.405} C_VEL
LIN {X 0,Y 389.494,Z 691.326,A -85,B 0,C 180,E1 -12148.837,E2 -12148.837} C_VEL
LIN {X 0,Y 391.031,Z 678.581,A -85,B 0,C 180,E1 -12150.129,E2 -12150.129} C_VEL
LIN {X 0,Y 392.501,Z 664.588,A -85,B 0,C 180,E1 -12151.283,E2 -12151.283} C_VEL
LIN {X 0,Y 392.586,Z 663.748,A -85,B 0,C 180,E1 -12151.344,E2 -12151.344} C_VEL
LIN {X 0,Y 392.501,Z 658.523,A -85,B 0,C 180,E1 -12151.749,E2 -12151.749} C_VEL
LIN {X 0,Y 390.538,Z 650.046,A -85,B 0,C 180,E1 -12152.451,E2 -12152.451} C_VEL
LIN {X 0,Y 388.565,Z 641.358,A -85,B 0,C 180,E1 -12153.084,E2 -12153.084} C_VEL
LIN {X 0,Y 388.365,Z 635.811,A -85,B 0,C 180,E1 -12153.375,E2 -12153.375} C_VEL
LIN {X 0,Y 389.188,Z 621.035,A -85,B 0,C 180,E1 -12153.916,E2 -12153.916} C_VEL
LIN {X 0,Y 389.72,Z 604.699,A -85,B 0,C 180,E1 -12154.299,E2 -12154.299} C_VEL
LIN {X 0,Y 392.505,Z 483.974,A -85,B 0,C 180,E1 -12156.572,E2 -12156.572} C_VEL
LIN {X 0,Y 382.409,Z 460.677,A -85,B 0,C 180,E1 -12157.87,E2 -12157.87} C_VEL
LIN {X 0,Y 377.826,Z 450.736,A -85,B 0,C 180,E1 -12158.505,E2 -12158.505} C_VEL
LIN {X 0,Y 376.093,Z 444.253,A -85,B 0,C 180,E1 -12160.158,E2 -12160.158} C_VEL
LIN {X 0,Y 376.094,Z 444.261,A -85,B 0,C 180,E1 -12163.658,E2 -12163.658} C_VEL
LIN {X 0,Y 376.049,Z 444.267,A -85,B 0,C 180,E1 -12167.608,E2 -12167.608} C_VEL
LIN {X 0,Y 376.01,Z 444.269,A -85,B 0,C 180,E1 -12170.844,E2 -12170.844} C_VEL
LIN {X 0,Y 375.998,Z 444.267,A -85,B 0,C 180,E1 -12174.282,E2 -12174.282} C_VEL
LIN {X 0,Y 376.023,Z 444.269,A -85,B 0,C 180,E1 -12176.652,E2 -12176.652} C_VEL
LIN {X 0,Y 375.98,Z 444.27,A -85,B 0,C 180,E1 -12179.079,E2 -12179.079} C_VEL
LIN {X 0,Y 375.955,Z 444.267,A -85,B 0,C 180,E1 -12182.828,E2 -12182.828} C_VEL
LIN {X 0,Y 375.961,Z 444.281,A -85,B 0,C 180,E1 -12185.415,E2 -12185.415} C_VEL
LIN {X 0,Y 375.979,Z 444.265,A -85,B 0,C 180,E1 -12188.271,E2 -12188.271} C_VEL
LIN {X 0,Y 375.948,Z 444.281,A -85,B 0,C 180,E1 -12191.602,E2 -12191.602} C_VEL
LIN {X 0,Y 375.931,Z 444.281,A -85,B 0,C 180,E1 -12195.268,E2 -12195.268} C_VEL
LIN {X 0,Y 375.962,Z 444.267,A -85,B 0,C 180,E1 -12198.395,E2 -12198.395} C_VEL
LIN {X 0,Y 375.98,Z 444.277,A -85,B 0,C 180,E1 -12201.729,E2 -12201.729} C_VEL
LIN {X 0,Y 375.982,Z 444.269,A -85,B 0,C 180,E1 -12205.332,E2 -12205.332} C_VEL
LIN {X 0,Y 375.959,Z 444.273,A -85,B 0,C 180,E1 -12208.438,E2 -12208.438} C_VEL
LIN {X 0,Y 375.985,Z 444.274,A -85,B 0,C 180,E1 -12212.14,E2 -12212.14} C_VEL
LIN {X 0,Y 376.007,Z 444.268,A -85,B 0,C 180,E1 -12214.539,E2 -12214.539} C_VEL
LIN {X 0,Y 375.959,Z 444.274,A -85,B 0,C 180,E1 -12218.045,E2 -12218.045} C_VEL
LIN {X 0,Y 376.025,Z 444.269,A -85,B 0,C 180,E1 -12221.474,E2 -12221.474} C_VEL
LIN {X 0,Y 376.059,Z 444.257,A -85,B 0,C 180,E1 -12224.832,E2 -12224.832} C_VEL
LIN {X 0,Y 376.05,Z 444.262,A -85,B 0,C 180,E1 -12228.136,E2 -12228.136} C_VEL
LIN {X 0,Y 376.258,Z 444.236,A -85,B 0,C 180,E1 -12231.877,E2 -12231.877} C_VEL
LIN {X 0,Y 376.172,Z 444.248,A -85,B 0,C 180,E1 -12234.64,E2 -12234.64} C_VEL
LIN {X 0,Y 376.352,Z 444.219,A -85,B 0,C 180,E1 -12237.859,E2 -12237.859} C_VEL
LIN {X 0,Y 376.489,Z 444.214,A -85,B 0,C 180,E1 -12240,E2 -12240} C_VEL
LIN {X 0,Y 376.189,Z 444.24,A -85,B 0,C 180,E1 -12243.213,E2 -12243.213} C_VEL
LIN {X 0,Y 376.247,Z 444.237,A -85,B 0,C 180,E1 -12246.435,E2 -12246.435} C_VEL
LIN {X 0,Y 376.205,Z 444.245,A -85,B 0,C 180,E1 -12248.595,E2 -12248.595} C_VEL
LIN {X 0,Y 376.049,Z 444.252,A -85,B 0,C 180,E1 -12251.863,E2 -12251.863} C_VEL
LIN {X 0,Y 376.058,Z 444.265,A -85,B 0,C 180,E1 -12255.167,E2 -12255.167} C_VEL
LIN {X 0,Y 376.009,Z 444.256,A -85,B 0,C 180,E1 -12258.527,E2 -12258.527} C_VEL
LIN {X 0,Y 375.963,Z 444.278,A -85,B 0,C 180,E1 -12261.954,E2 -12261.954} C_VEL
LIN {X 0,Y 376.006,Z 444.273,A -85,B 0,C 180,E1 -12265.461,E2 -12265.461} C_VEL
LIN {X 0,Y 375.976,Z 444.273,A -85,B 0,C 180,E1 -12269.078,E2 -12269.078} C_VEL
LIN {X 0,Y 375.951,Z 444.277,A -85,B 0,C 180,E1 -12272.828,E2 -12272.828} C_VEL
LIN {X 0,Y 375.958,Z 444.28,A -85,B 0,C 180,E1 -12275.415,E2 -12275.415} C_VEL
LIN {X 0,Y 375.976,Z 444.276,A -85,B 0,C 180,E1 -12278.271,E2 -12278.271} C_VEL
LIN {X 0,Y 375.935,Z 444.284,A -85,B 0,C 180,E1 -12281.601,E2 -12281.601} C_VEL
LIN {X 0,Y 375.979,Z 444.277,A -85,B 0,C 180,E1 -12285.26,E2 -12285.26} C_VEL
LIN {X 0,Y 375.988,Z 444.276,A -85,B 0,C 180,E1 -12288.39,E2 -12288.39} C_VEL
LIN {X 0,Y 375.964,Z 444.282,A -85,B 0,C 180,E1 -12291.911,E2 -12291.911} C_VEL
LIN {X 0,Y 376.014,Z 444.322,A -85,B 0,C 180,E1 -12294.22,E2 -12294.22} C_VEL
LIN {X 0,Y 379.507,Z 457.773,A -85,B 0,C 180,E1 -12297.286,E2 -12297.286} C_VEL
LIN {X 0,Y 382.571,Z 470.375,A -85,B 0,C 180,E1 -12299.963,E2 -12299.963} C_VEL
LIN {X 0,Y 386.329,Z 479.692,A -85,B 0,C 180,E1 -12300.466,E2 -12300.466} C_VEL
LIN {X 0,Y 392.076,Z 509.965,A -85,B 0,C 180,E1 -12301.547,E2 -12301.547} C_VEL
LIN {X 0,Y 389.519,Z 622.086,A -85,B 0,C 180,E1 -12303.657,E2 -12303.657} C_VEL
LIN {X 0,Y 388.941,Z 641.145,A -85,B 0,C 180,E1 -12304.083,E2 -12304.083} C_VEL
LIN {X 0,Y 387.934,Z 656.424,A -85,B 0,C 180,E1 -12304.623,E2 -12304.623} C_VEL
LIN {X 0,Y 386.771,Z 671.161,A -85,B 0,C 180,E1 -12305.361,E2 -12305.361} C_VEL
LIN {X 0,Y 385.472,Z 684.499,A -85,B 0,C 180,E1 -12306.226,E2 -12306.226} C_VEL
LIN {X 0,Y 383.976,Z 697.31,A -85,B 0,C 180,E1 -12307.253,E2 -12307.253} C_VEL
LIN {X 0,Y 382.344,Z 710.63,A -85,B 0,C 180,E1 -12308.572,E2 -12308.572} C_VEL
LIN {X 0,Y 380.697,Z 722.781,A -85,B 0,C 180,E1 -12310.03,E2 -12310.03} C_VEL
LIN {X 0,Y 379.307,Z 733.888,A -85,B 0,C 180,E1 -12311.64,E2 -12311.64} C_VEL
LIN {X 0,Y 377.975,Z 743.275,A -85,B 0,C 180,E1 -12313.249,E2 -12313.249} C_VEL
LIN {X 0,Y 376.783,Z 752.466,A -85,B 0,C 180,E1 -12315.139,E2 -12315.139} C_VEL
LIN {X 0,Y 375.911,Z 760.097,A -85,B 0,C 180,E1 -12317.035,E2 -12317.035} C_VEL
LIN {X 0,Y 375.394,Z 765.595,A -85,B 0,C 180,E1 -12318.663,E2 -12318.663} C_VEL
LIN {X 0,Y 374.845,Z 771.575,A -85,B 0,C 180,E1 -12320.829,E2 -12320.829} C_VEL
LIN {X 0,Y 374.656,Z 775.119,A -85,B 0,C 180,E1 -12322.454,E2 -12322.454} C_VEL
LIN {X 0,Y 374.502,Z 778.726,A -85,B 0,C 180,E1 -12324.615,E2 -12324.615} C_VEL
LIN {X 0,Y 374.437,Z 781.108,A -85,B 0,C 180,E1 -12326.771,E2 -12326.771} C_VEL
LIN {X 0,Y 374.513,Z 782.322,A -85,B 0,C 180,E1 -12328.924,E2 -12328.924} C_VEL
LIN {X 0,Y 374.513,Z 782.329,A -85,B 0,C 180,E1 -12331.075,E2 -12331.075} C_VEL
LIN {X 0,Y 374.444,Z 781.172,A -85,B 0,C 180,E1 -12333.227,E2 -12333.227} C_VEL
LIN {X 0,Y 374.502,Z 778.858,A -85,B 0,C 180,E1 -12335.383,E2 -12335.383} C_VEL
LIN {X 0,Y 374.657,Z 775.336,A -85,B 0,C 180,E1 -12337.545,E2 -12337.545} C_VEL
LIN {X 0,Y 374.963,Z 770.52,A -85,B 0,C 180,E1 -12339.711,E2 -12339.711} C_VEL
LIN {X 0,Y 375.583,Z 764.288,A -85,B 0,C 180,E1 -12341.878,E2 -12341.878} C_VEL
LIN {X 0,Y 376.386,Z 756.463,A -85,B 0,C 180,E1 -12344.048,E2 -12344.048} C_VEL
LIN {X 0,Y 377.465,Z 748.146,A -85,B 0,C 180,E1 -12345.939,E2 -12345.939} C_VEL
LIN {X 0,Y 378.847,Z 738.146,A -85,B 0,C 180,E1 -12347.823,E2 -12347.823} C_VEL
LIN {X 0,Y 380.438,Z 726.843,A -85,B 0,C 180,E1 -12349.585,E2 -12349.585} C_VEL
LIN {X 0,Y 382.125,Z 714.655,A -85,B 0,C 180,E1 -12351.157,E2 -12351.157} C_VEL
LIN {X 0,Y 383.787,Z 702.295,A -85,B 0,C 180,E1 -12352.473,E2 -12352.473} C_VEL
LIN {X 0,Y 385.439,Z 688.813,A -85,B 0,C 180,E1 -12353.649,E2 -12353.649} C_VEL
LIN {X 0,Y 387.031,Z 673.911,A -85,B 0,C 180,E1 -12354.685,E2 -12354.685} C_VEL
LIN {X 0,Y 388.362,Z 658.473,A -85,B 0,C 180,E1 -12355.504,E2 -12355.504} C_VEL
LIN {X 0,Y 389.509,Z 642.715,A -85,B 0,C 180,E1 -12356.09,E2 -12356.09} C_VEL
LIN {X 0,Y 390.214,Z 626.716,A -85,B 0,C 180,E1 -12356.471,E2 -12356.471} C_VEL
LIN {X 0,Y 392.995,Z 510.407,A -85,B 0,C 180,E1 -12358.678,E2 -12358.678} C_VEL
LIN {X 0,Y 389.018,Z 488.757,A -85,B 0,C 180,E1 -12359.477,E2 -12359.477} C_VEL
LIN {X 0,Y 386.967,Z 479.573,A -85,B 0,C 180,E1 -12359.856,E2 -12359.856} C_VEL
LIN {X 0,Y 382.488,Z 469.278,A -85,B 0,C 180,E1 -12360.504,E2 -12360.504} C_VEL
LIN {X 0,Y 379.525,Z 457.299,A -85,B 0,C 180,E1 -12363.2,E2 -12363.2} C_VEL
LIN {X 0,Y 376.8,Z 447.227,A -85,B 0,C 180,E1 -12365.605,E2 -12365.605} C_VEL
LIN {X 0,Y 375.988,Z 444.279,A -85,B 0,C 180,E1 -12366.344,E2 -12366.344} C_VEL
LIN {X 0,Y 375.995,Z 444.269,A -85,B 0,C 180,E1 -12369.972,E2 -12369.972} C_VEL
LIN {X 0,Y 375.983,Z 444.269,A -85,B 0,C 180,E1 -12373.198,E2 -12373.198} C_VEL
LIN {X 0,Y 375.93,Z 444.273,A -85,B 0,C 180,E1 -12376.81,E2 -12376.81} C_VEL
LIN {X 0,Y 375.958,Z 444.282,A -85,B 0,C 180,E1 -12380.537,E2 -12380.537} C_VEL
LIN {X 0,Y 375.959,Z 444.278,A -85,B 0,C 180,E1 -12383.495,E2 -12383.495} C_VEL
LIN {X 0,Y 375.956,Z 444.28,A -85,B 0,C 180,E1 -12385.888,E2 -12385.888} C_VEL
LIN {X 0,Y 375.957,Z 444.276,A -85,B 0,C 180,E1 -12389.687,E2 -12389.687} C_VEL
LIN {X 0,Y 376.013,Z 444.267,A -85,B 0,C 180,E1 -12393.348,E2 -12393.348} C_VEL
LIN {X 0,Y 375.989,Z 444.274,A -85,B 0,C 180,E1 -12396.888,E2 -12396.888} C_VEL
LIN {X 0,Y 375.99,Z 444.272,A -85,B 0,C 180,E1 -12400.339,E2 -12400.339} C_VEL
LIN {X 0,Y 376.021,Z 444.264,A -85,B 0,C 180,E1 -12403.719,E2 -12403.719} C_VEL
LIN {X 0,Y 376.099,Z 444.256,A -85,B 0,C 180,E1 -12407.042,E2 -12407.042} C_VEL
LIN {X 0,Y 376.117,Z 444.254,A -85,B 0,C 180,E1 -12410.319,E2 -12410.319} C_VEL
LIN {X 0,Y 376.223,Z 444.247,A -85,B 0,C 180,E1 -12412.487,E2 -12412.487} C_VEL
LIN {X 0,Y 376.165,Z 444.25,A -85,B 0,C 180,E1 -12414.64,E2 -12414.64} C_VEL
LIN {X 0,Y 376.347,Z 444.224,A -85,B 0,C 180,E1 -12417.86,E2 -12417.86} C_VEL
LIN {X 0,Y 376.481,Z 444.215,A -85,B 0,C 180,E1 -12420,E2 -12420} C_VEL
LIN {X 0,Y 376.185,Z 444.249,A -85,B 0,C 180,E1 -12423.213,E2 -12423.213} C_VEL
LIN {X 0,Y 376.229,Z 444.246,A -85,B 0,C 180,E1 -12426.604,E2 -12426.604} C_VEL
LIN {X 0,Y 376.198,Z 444.247,A -85,B 0,C 180,E1 -12428.596,E2 -12428.596} C_VEL
LIN {X 0,Y 376.043,Z 444.265,A -85,B 0,C 180,E1 -12431.864,E2 -12431.864} C_VEL
LIN {X 0,Y 376.055,Z 444.266,A -85,B 0,C 180,E1 -12435.168,E2 -12435.168} C_VEL
LIN {X 0,Y 376.018,Z 444.272,A -85,B 0,C 180,E1 -12438.527,E2 -12438.527} C_VEL
LIN {X 0,Y 375.959,Z 444.279,A -85,B 0,C 180,E1 -12441.955,E2 -12441.955} C_VEL
LIN {X 0,Y 376.001,Z 444.276,A -85,B 0,C 180,E1 -12445.462,E2 -12445.462} C_VEL
LIN {X 0,Y 375.972,Z 444.277,A -85,B 0,C 180,E1 -12449.079,E2 -12449.079} C_VEL
LIN {X 0,Y 375.953,Z 444.275,A -85,B 0,C 180,E1 -12452.828,E2 -12452.828} C_VEL
LIN {X 0,Y 376.023,Z 444.457,A -85,B 0,C 180,E1 -12455.235,E2 -12455.235} C_VEL
LIN {X 0,Y 377.955,Z 451.669,A -85,B 0,C 180,E1 -12457.135,E2 -12457.135} C_VEL
LIN {X 0,Y 386.794,Z 469.605,A -85,B 0,C 180,E1 -12458.366,E2 -12458.366} C_VEL
LIN {X 0,Y 393.535,Z 485.342,A -85,B 0,C 180,E1 -12459.293,E2 -12459.293} C_VEL
LIN {X 0,Y 390.185,Z 616.758,A -85,B 0,C 180,E1 -12461.811,E2 -12461.811} C_VEL
LIN {X 0,Y 389.366,Z 632.199,A -85,B 0,C 180,E1 -12462.314,E2 -12462.314} C_VEL
LIN {X 0,Y 388.338,Z 646.142,A -85,B 0,C 180,E1 -12462.962,E2 -12462.962} C_VEL
LIN {X 0,Y 386.994,Z 661.094,A -85,B 0,C 180,E1 -12463.886,E2 -12463.886} C_VEL
LIN {X 0,Y 385.381,Z 675.589,A -85,B 0,C 180,E1 -12465.032,E2 -12465.032} C_VEL
LIN {X 0,Y 383.821,Z 688.271,A -85,B 0,C 180,E1 -12466.274,E2 -12466.274} C_VEL
LIN {X 0,Y 382.031,Z 701.206,A -85,B 0,C 180,E1 -12467.821,E2 -12467.821} C_VEL
LIN {X 0,Y 380.454,Z 712.407,A -85,B 0,C 180,E1 -12469.446,E2 -12469.446} C_VEL
LIN {X 0,Y 378.929,Z 722.328,A -85,B 0,C 180,E1 -12471.167,E2 -12471.167} C_VEL
LIN {X 0,Y 377.597,Z 731.802,A -85,B 0,C 180,E1 -12473.163,E2 -12473.163} C_VEL
LIN {X 0,Y 376.529,Z 739.766,A -85,B 0,C 180,E1 -12475.213,E2 -12475.213} C_VEL
LIN {X 0,Y 375.647,Z 746.451,A -85,B 0,C 180,E1 -12477.343,E2 -12477.343} C_VEL
LIN {X 0,Y 375.083,Z 751.994,A -85,B 0,C 180,E1 -12479.61,E2 -12479.61} C_VEL
LIN {X 0,Y 374.609,Z 756.056,A -85,B 0,C 180,E1 -12481.856,E2 -12481.856} C_VEL
LIN {X 0,Y 374.382,Z 758.993,A -85,B 0,C 180,E1 -12484.3,E2 -12484.3} C_VEL
LIN {X 0,Y 374.258,Z 760.449,A -85,B 0,C 180,E1 -12486.776,E2 -12486.776} C_VEL
LIN {X 0,Y 374.252,Z 760.443,A -85,B 0,C 180,E1 -12489.097,E2 -12489.097} C_VEL
LIN {X 0,Y 374.359,Z 759.135,A -85,B 0,C 180,E1 -12491.389,E2 -12491.389} C_VEL
LIN {X 0,Y 374.614,Z 756.552,A -85,B 0,C 180,E1 -12493.656,E2 -12493.656} C_VEL
LIN {X 0,Y 374.963,Z 752.683,A -85,B 0,C 180,E1 -12495.898,E2 -12495.898} C_VEL
LIN {X 0,Y 375.444,Z 747.481,A -85,B 0,C 180,E1 -12498.118,E2 -12498.118} C_VEL
LIN {X 0,Y 376.19,Z 740.822,A -85,B 0,C 180,E1 -12500.321,E2 -12500.321} C_VEL
LIN {X 0,Y 377.097,Z 733.619,A -85,B 0,C 180,E1 -12502.241,E2 -12502.241} C_VEL
LIN {X 0,Y 378.232,Z 725.03,A -85,B 0,C 180,E1 -12504.135,E2 -12504.135} C_VEL
LIN {X 0,Y 379.73,Z 714.499,A -85,B 0,C 180,E1 -12506.047,E2 -12506.047} C_VEL
LIN {X 0,Y 381.155,Z 704.077,A -85,B 0,C 180,E1 -12507.623,E2 -12507.623} C_VEL
LIN {X 0,Y 382.667,Z 692.57,A -85,B 0,C 180,E1 -12509.08,E2 -12509.08} C_VEL
LIN {X 0,Y 384.248,Z 680.044,A -85,B 0,C 180,E1 -12510.394,E2 -12510.394} C_VEL
LIN {X 0,Y 385.772,Z 666.34,A -85,B 0,C 180,E1 -12511.566,E2 -12511.566} C_VEL
LIN {X 0,Y 387.118,Z 652.148,A -85,B 0,C 180,E1 -12512.534,E2 -12512.534} C_VEL
LIN {X 0,Y 388.165,Z 638.839,A -85,B 0,C 180,E1 -12513.244,E2 -12513.244} C_VEL
LIN {X 0,Y 388.365,Z 635.811,A -85,B 0,C 180,E1 -12513.375,E2 -12513.375} C_VEL
LIN {X 0,Y 388.192,Z 630.185,A -85,B 0,C 180,E1 -12513.644,E2 -12513.644} C_VEL
LIN {X 0,Y 384.093,Z 613.757,A -85,B 0,C 180,E1 -12514.491,E2 -12514.491} C_VEL
LIN {X 0,Y 383.316,Z 608.047,A -85,B 0,C 180,E1 -12514.685,E2 -12514.685} C_VEL
LIN {X 0,Y 383.281,Z 606.1,A -85,B 0,C 180,E1 -12514.728,E2 -12514.728} C_VEL
LIN {X 0,Y 386.253,Z 485.923,A -85,B 0,C 180,E1 -12517.02,E2 -12517.02} C_VEL
LIN {X 0,Y 376.254,Z 463.063,A -85,B 0,C 180,E1 -12518.336,E2 -12518.336} C_VEL
LIN {X 0,Y 370.588,Z 450.989,A -85,B 0,C 180,E1 -12519.125,E2 -12519.125} C_VEL
LIN {X 0,Y 369.047,Z 445.127,A -85,B 0,C 180,E1 -12520.632,E2 -12520.632} C_VEL
LIN {X 0,Y 369.02,Z 445.145,A -85,B 0,C 180,E1 -12524.335,E2 -12524.335} C_VEL
LIN {X 0,Y 369.005,Z 445.143,A -85,B 0,C 180,E1 -12527.769,E2 -12527.769} C_VEL
LIN {X 0,Y 368.945,Z 445.149,A -85,B 0,C 180,E1 -12531.219,E2 -12531.219} C_VEL
LIN {X 0,Y 368.962,Z 445.143,A -85,B 0,C 180,E1 -12534.775,E2 -12534.775} C_VEL
LIN {X 0,Y 368.99,Z 445.139,A -85,B 0,C 180,E1 -12538.436,E2 -12538.436} C_VEL
LIN {X 0,Y 368.903,Z 445.146,A -85,B 0,C 180,E1 -12542.238,E2 -12542.238} C_VEL
LIN {X 0,Y 368.933,Z 445.154,A -85,B 0,C 180,E1 -12545.002,E2 -12545.002} C_VEL
LIN {X 0,Y 368.914,Z 445.145,A -85,B 0,C 180,E1 -12548.641,E2 -12548.641} C_VEL
LIN {X 0,Y 368.891,Z 445.155,A -85,B 0,C 180,E1 -12552.01,E2 -12552.01} C_VEL
LIN {X 0,Y 368.884,Z 445.158,A -85,B 0,C 180,E1 -12555.176,E2 -12555.176} C_VEL
LIN {X 0,Y 368.912,Z 445.145,A -85,B 0,C 180,E1 -12558.181,E2 -12558.181} C_VEL
LIN {X 0,Y 368.915,Z 445.157,A -85,B 0,C 180,E1 -12561.359,E2 -12561.359} C_VEL
LIN {X 0,Y 368.939,Z 445.144,A -85,B 0,C 180,E1 -12565.146,E2 -12565.146} C_VEL
LIN {X 0,Y 368.931,Z 445.149,A -85,B 0,C 180,E1 -12569.046,E2 -12569.046} C_VEL
LIN {X 0,Y 368.965,Z 445.147,A -85,B 0,C 180,E1 -12572.796,E2 -12572.796} C_VEL
LIN {X 0,Y 368.938,Z 445.138,A -85,B 0,C 180,E1 -12576.116,E2 -12576.116} C_VEL
LIN {X 0,Y 368.938,Z 445.154,A -85,B 0,C 180,E1 -12579.947,E2 -12579.947} C_VEL
LIN {X 0,Y 368.976,Z 445.135,A -85,B 0,C 180,E1 -12583.398,E2 -12583.398} C_VEL
LIN {X 0,Y 369.058,Z 445.135,A -85,B 0,C 180,E1 -12586.79,E2 -12586.79} C_VEL
LIN {X 0,Y 369.068,Z 445.122,A -85,B 0,C 180,E1 -12590.131,E2 -12590.131} C_VEL
LIN {X 0,Y 369.189,Z 445.118,A -85,B 0,C 180,E1 -12592.342,E2 -12592.342} C_VEL
LIN {X 0,Y 369.145,Z 445.124,A -85,B 0,C 180,E1 -12594.537,E2 -12594.537} C_VEL
LIN {X 0,Y 369.317,Z 445.095,A -85,B 0,C 180,E1 -12597.819,E2 -12597.819} C_VEL
LIN {X 0,Y 369.458,Z 445.089,A -85,B 0,C 180,E1 -12600,E2 -12600} C_VEL
LIN {X 0,Y 369.319,Z 445.099,A -85,B 0,C 180,E1 -12602.181,E2 -12602.181} C_VEL
LIN {X 0,Y 369.208,Z 445.113,A -85,B 0,C 180,E1 -12606.558,E2 -12606.558} C_VEL
LIN {X 0,Y 369.138,Z 445.126,A -85,B 0,C 180,E1 -12608.761,E2 -12608.761} C_VEL
LIN {X 0,Y 369.004,Z 445.129,A -85,B 0,C 180,E1 -12612.093,E2 -12612.093} C_VEL
LIN {X 0,Y 368.997,Z 445.147,A -85,B 0,C 180,E1 -12615.465,E2 -12615.465} C_VEL
LIN {X 0,Y 368.958,Z 445.134,A -85,B 0,C 180,E1 -12618.894,E2 -12618.894} C_VEL
LIN {X 0,Y 368.932,Z 445.151,A -85,B 0,C 180,E1 -12622.395,E2 -12622.395} C_VEL
LIN {X 0,Y 369,Z 445.145,A -85,B 0,C 180,E1 -12625.98,E2 -12625.98} C_VEL
LIN {X 0,Y 368.967,Z 445.146,A -85,B 0,C 180,E1 -12628.813,E2 -12628.813} C_VEL
LIN {X 0,Y 368.899,Z 445.157,A -85,B 0,C 180,E1 -12632.238,E2 -12632.238} C_VEL
LIN {X 0,Y 368.929,Z 445.153,A -85,B 0,C 180,E1 -12635.001,E2 -12635.001} C_VEL
LIN {X 0,Y 368.91,Z 445.155,A -85,B 0,C 180,E1 -12638.64,E2 -12638.64} C_VEL
LIN {X 0,Y 368.881,Z 445.16,A -85,B 0,C 180,E1 -12642.009,E2 -12642.009} C_VEL
LIN {X 0,Y 368.954,Z 445.152,A -85,B 0,C 180,E1 -12645.187,E2 -12645.187} C_VEL
LIN {X 0,Y 368.94,Z 445.153,A -85,B 0,C 180,E1 -12648.185,E2 -12648.185} C_VEL
LIN {X 0,Y 368.909,Z 445.157,A -85,B 0,C 180,E1 -12651.359,E2 -12651.359} C_VEL
LIN {X 0,Y 368.964,Z 445.321,A -85,B 0,C 180,E1 -12653.726,E2 -12653.726} C_VEL
LIN {X 0,Y 372.464,Z 458.553,A -85,B 0,C 180,E1 -12656.825,E2 -12656.825} C_VEL
LIN {X 0,Y 375.221,Z 469.892,A -85,B 0,C 180,E1 -12659.336,E2 -12659.336} C_VEL
LIN {X 0,Y 380.355,Z 482.343,A -85,B 0,C 180,E1 -12660.039,E2 -12660.039} C_VEL
LIN {X 0,Y 385.707,Z 510.724,A -85,B 0,C 180,E1 -12661.073,E2 -12661.073} C_VEL
LIN {X 0,Y 383.434,Z 608.494,A -85,B 0,C 180,E1 -12662.948,E2 -12662.948} C_VEL
LIN {X 0,Y 382.65,Z 637.995,A -85,B 0,C 180,E1 -12663.551,E2 -12663.551} C_VEL
LIN {X 0,Y 381.706,Z 653.481,A -85,B 0,C 180,E1 -12664.069,E2 -12664.069} C_VEL
LIN {X 0,Y 380.595,Z 667.311,A -85,B 0,C 180,E1 -12664.721,E2 -12664.721} C_VEL
LIN {X 0,Y 379.213,Z 681.237,A -85,B 0,C 180,E1 -12665.583,E2 -12665.583} C_VEL
LIN {X 0,Y 377.552,Z 695.438,A -85,B 0,C 180,E1 -12666.699,E2 -12666.699} C_VEL
LIN {X 0,Y 375.807,Z 709.062,A -85,B 0,C 180,E1 -12668.036,E2 -12668.036} C_VEL
LIN {X 0,Y 374.12,Z 721.438,A -85,B 0,C 180,E1 -12669.52,E2 -12669.52} C_VEL
LIN {X 0,Y 372.893,Z 730.635,A -85,B 0,C 180,E1 -12670.837,E2 -12670.837} C_VEL
LIN {X 0,Y 371.277,Z 741.459,A -85,B 0,C 180,E1 -12672.654,E2 -12672.654} C_VEL
LIN {X 0,Y 369.996,Z 750.926,A -85,B 0,C 180,E1 -12674.578,E2 -12674.578} C_VEL
LIN {X 0,Y 368.917,Z 759.823,A -85,B 0,C 180,E1 -12676.785,E2 -12676.785} C_VEL
LIN {X 0,Y 368.157,Z 766.967,A -85,B 0,C 180,E1 -12678.994,E2 -12678.994} C_VEL
LIN {X 0,Y 367.727,Z 772.591,A -85,B 0,C 180,E1 -12681.205,E2 -12681.205} C_VEL
LIN {X 0,Y 367.481,Z 776.85,A -85,B 0,C 180,E1 -12683.41,E2 -12683.41} C_VEL
LIN {X 0,Y 367.399,Z 779.846,A -85,B 0,C 180,E1 -12685.611,E2 -12685.611} C_VEL
LIN {X 0,Y 367.349,Z 781.646,A -85,B 0,C 180,E1 -12687.807,E2 -12687.807} C_VEL
LIN {X 0,Y 367.454,Z 782.268,A -85,B 0,C 180,E1 -12689.999,E2 -12689.999} C_VEL
LIN {X 0,Y 367.351,Z 781.69,A -85,B 0,C 180,E1 -12692.192,E2 -12692.192} C_VEL
LIN {X 0,Y 367.405,Z 779.967,A -85,B 0,C 180,E1 -12694.388,E2 -12694.388} C_VEL
LIN {X 0,Y 367.481,Z 777.065,A -85,B 0,C 180,E1 -12696.588,E2 -12696.588} C_VEL
LIN {X 0,Y 367.729,Z 772.919,A -85,B 0,C 180,E1 -12698.794,E2 -12698.794} C_VEL
LIN {X 0,Y 368.159,Z 767.421,A -85,B 0,C 180,E1 -12701.004,E2 -12701.004} C_VEL
LIN {X 0,Y 368.713,Z 762.29,A -85,B 0,C 180,E1 -12702.661,E2 -12702.661} C_VEL
LIN {X 0,Y 369.57,Z 755.181,A -85,B 0,C 180,E1 -12704.593,E2 -12704.593} C_VEL
LIN {X 0,Y 370.743,Z 746.648,A -85,B 0,C 180,E1 -12706.519,E2 -12706.519} C_VEL
LIN {X 0,Y 372.051,Z 738.011,A -85,B 0,C 180,E1 -12708.16,E2 -12708.16} C_VEL
LIN {X 0,Y 373.805,Z 726.117,A -85,B 0,C 180,E1 -12710.037,E2 -12710.037} C_VEL
LIN {X 0,Y 375.462,Z 714.573,A -85,B 0,C 180,E1 -12711.551,E2 -12711.551} C_VEL
LIN {X 0,Y 377.196,Z 702.245,A -85,B 0,C 180,E1 -12712.888,E2 -12712.888} C_VEL
LIN {X 0,Y 378.94,Z 688.813,A -85,B 0,C 180,E1 -12714.08,E2 -12714.08} C_VEL
LIN {X 0,Y 380.579,Z 673.982,A -85,B 0,C 180,E1 -12715.133,E2 -12715.133} C_VEL
LIN {X 0,Y 381.985,Z 658.667,A -85,B 0,C 180,E1 -12715.961,E2 -12715.961} C_VEL
LIN {X 0,Y 383.159,Z 643.125,A -85,B 0,C 180,E1 -12716.556,E2 -12716.556} C_VEL
LIN {X 0,Y 383.896,Z 627.481,A -85,B 0,C 180,E1 -12716.942,E2 -12716.942} C_VEL
LIN {X 0,Y 386.833,Z 511.437,A -85,B 0,C 180,E1 -12719.176,E2 -12719.176} C_VEL
LIN {X 0,Y 382.615,Z 488.636,A -85,B 0,C 180,E1 -12720.048,E2 -12720.048} C_VEL
LIN {X 0,Y 381.196,Z 482.44,A -85,B 0,C 180,E1 -12720.315,E2 -12720.315} C_VEL
LIN {X 0,Y 375.248,Z 468.997,A -85,B 0,C 180,E1 -12721.202,E2 -12721.202} C_VEL
LIN {X 0,Y 371.606,Z 454.638,A -85,B 0,C 180,E1 -12724.566,E2 -12724.566} C_VEL
LIN {X 0,Y 368.901,Z 445.155,A -85,B 0,C 180,E1 -12727.013,E2 -12727.013} C_VEL
LIN {X 0,Y 368.948,Z 445.147,A -85,B 0,C 180,E1 -12730.364,E2 -12730.364} C_VEL
LIN {X 0,Y 368.925,Z 445.15,A -85,B 0,C 180,E1 -12733.623,E2 -12733.623} C_VEL
LIN {X 0,Y 368.883,Z 445.151,A -85,B 0,C 180,E1 -12736.696,E2 -12736.696} C_VEL
LIN {X 0,Y 368.906,Z 445.157,A -85,B 0,C 180,E1 -12739.642,E2 -12739.642} C_VEL
LIN {X 0,Y 368.897,Z 445.158,A -85,B 0,C 180,E1 -12743.143,E2 -12743.143} C_VEL
LIN {X 0,Y 368.892,Z 445.157,A -85,B 0,C 180,E1 -12746.462,E2 -12746.462} C_VEL
LIN {X 0,Y 368.922,Z 445.153,A -85,B 0,C 180,E1 -12749.046,E2 -12749.046} C_VEL
LIN {X 0,Y 368.956,Z 445.146,A -85,B 0,C 180,E1 -12752.796,E2 -12752.796} C_VEL
LIN {X 0,Y 368.938,Z 445.149,A -85,B 0,C 180,E1 -12756.113,E2 -12756.113} C_VEL
LIN {X 0,Y 368.929,Z 445.148,A -85,B 0,C 180,E1 -12759.947,E2 -12759.947} C_VEL
LIN {X 0,Y 368.968,Z 445.142,A -85,B 0,C 180,E1 -12763.399,E2 -12763.399} C_VEL
LIN {X 0,Y 369.052,Z 445.133,A -85,B 0,C 180,E1 -12766.79,E2 -12766.79} C_VEL
LIN {X 0,Y 369.065,Z 445.133,A -85,B 0,C 180,E1 -12770.132,E2 -12770.132} C_VEL
LIN {X 0,Y 369.181,Z 445.126,A -85,B 0,C 180,E1 -12772.342,E2 -12772.342} C_VEL
LIN {X 0,Y 369.138,Z 445.124,A -85,B 0,C 180,E1 -12774.538,E2 -12774.538} C_VEL
LIN {X 0,Y 369.312,Z 445.1,A -85,B 0,C 180,E1 -12777.819,E2 -12777.819} C_VEL
LIN {X 0,Y 369.451,Z 445.091,A -85,B 0,C 180,E1 -12780,E2 -12780} C_VEL
LIN {X 0,Y 369.312,Z 445.102,A -85,B 0,C 180,E1 -12782.181,E2 -12782.181} C_VEL
LIN {X 0,Y 369.199,Z 445.122,A -85,B 0,C 180,E1 -12786.591,E2 -12786.591} C_VEL
LIN {X 0,Y 369.131,Z 445.129,A -85,B 0,C 180,E1 -12788.761,E2 -12788.761} C_VEL
LIN {X 0,Y 368.998,Z 445.144,A -85,B 0,C 180,E1 -12792.094,E2 -12792.094} C_VEL
LIN {X 0,Y 368.994,Z 445.146,A -85,B 0,C 180,E1 -12795.465,E2 -12795.465} C_VEL
LIN {X 0,Y 368.977,Z 445.146,A -85,B 0,C 180,E1 -12798.893,E2 -12798.893} C_VEL
LIN {X 0,Y 368.927,Z 445.159,A -85,B 0,C 180,E1 -12802.396,E2 -12802.396} C_VEL
LIN {X 0,Y 368.995,Z 445.143,A -85,B 0,C 180,E1 -12805.981,E2 -12805.981} C_VEL
LIN {X 0,Y 368.962,Z 445.152,A -85,B 0,C 180,E1 -12808.814,E2 -12808.814} C_VEL
LIN {X 0,Y 368.905,Z 445.153,A -85,B 0,C 180,E1 -12812.238,E2 -12812.238} C_VEL
LIN {X 0,Y 368.945,Z 445.25,A -85,B 0,C 180,E1 -12814.604,E2 -12814.604} C_VEL
LIN {X 0,Y 370.835,Z 452.161,A -85,B 0,C 180,E1 -12816.443,E2 -12816.443} C_VEL
LIN {X 0,Y 380.505,Z 471.274,A -85,B 0,C 180,E1 -12817.826,E2 -12817.826} C_VEL
LIN {X 0,Y 387.268,Z 486.897,A -85,B 0,C 180,E1 -12818.786,E2 -12818.786} C_VEL
LIN {X 0,Y 383.927,Z 616.69,A -85,B 0,C 180,E1 -12821.321,E2 -12821.321} C_VEL
LIN {X 0,Y 383.037,Z 632.336,A -85,B 0,C 180,E1 -12821.834,E2 -12821.834} C_VEL
LIN {X 0,Y 381.945,Z 646.663,A -85,B 0,C 180,E1 -12822.51,E2 -12822.51} C_VEL
LIN {X 0,Y 380.547,Z 661.496,A -85,B 0,C 180,E1 -12823.444,E2 -12823.444} C_VEL
LIN {X 0,Y 378.94,Z 675.511,A -85,B 0,C 180,E1 -12824.568,E2 -12824.568} C_VEL
LIN {X 0,Y 377.256,Z 688.626,A -85,B 0,C 180,E1 -12825.873,E2 -12825.873} C_VEL
LIN {X 0,Y 375.477,Z 700.727,A -85,B 0,C 180,E1 -12827.334,E2 -12827.334} C_VEL
LIN {X 0,Y 373.908,Z 711.245,A -85,B 0,C 180,E1 -12828.864,E2 -12828.864} C_VEL
LIN {X 0,Y 372.205,Z 721.986,A -85,B 0,C 180,E1 -12830.73,E2 -12830.73} C_VEL
LIN {X 0,Y 370.809,Z 731.534,A -85,B 0,C 180,E1 -12832.754,E2 -12832.754} C_VEL
LIN {X 0,Y 369.624,Z 739.605,A -85,B 0,C 180,E1 -12834.846,E2 -12834.846} C_VEL
LIN {X 0,Y 368.68,Z 746.342,A -85,B 0,C 180,E1 -12837.01,E2 -12837.01} C_VEL
LIN {X 0,Y 368.092,Z 751.751,A -85,B 0,C 180,E1 -12839.226,E2 -12839.226} C_VEL
LIN {X 0,Y 367.589,Z 756.041,A -85,B 0,C 180,E1 -12841.581,E2 -12841.581} C_VEL
LIN {X 0,Y 367.305,Z 759.056,A -85,B 0,C 180,E1 -12844.066,E2 -12844.066} C_VEL
LIN {X 0,Y 367.174,Z 760.659,A -85,B 0,C 180,E1 -12846.746,E2 -12846.746} C_VEL
LIN {X 0,Y 367.145,Z 760.716,A -85,B 0,C 180,E1 -12848.673,E2 -12848.673} C_VEL
LIN {X 0,Y 367.242,Z 759.651,A -85,B 0,C 180,E1 -12851.015,E2 -12851.015} C_VEL
LIN {X 0,Y 367.496,Z 757.31,A -85,B 0,C 180,E1 -12853.331,E2 -12853.331} C_VEL
LIN {X 0,Y 367.846,Z 753.687,A -85,B 0,C 180,E1 -12855.619,E2 -12855.619} C_VEL
LIN {X 0,Y 368.295,Z 748.744,A -85,B 0,C 180,E1 -12857.884,E2 -12857.884} C_VEL
LIN {X 0,Y 369.034,Z 742.358,A -85,B 0,C 180,E1 -12860.132,E2 -12860.132} C_VEL
LIN {X 0,Y 370.083,Z 734.356,A -85,B 0,C 180,E1 -12862.362,E2 -12862.362} C_VEL
LIN {X 0,Y 371.277,Z 725.841,A -85,B 0,C 180,E1 -12864.297,E2 -12864.297} C_VEL
LIN {X 0,Y 372.789,Z 715.593,A -85,B 0,C 180,E1 -12866.218,E2 -12866.218} C_VEL
LIN {X 0,Y 374.289,Z 705.15,A -85,B 0,C 180,E1 -12867.848,E2 -12867.848} C_VEL
LIN {X 0,Y 375.855,Z 693.81,A -85,B 0,C 180,E1 -12869.331,E2 -12869.331} C_VEL
LIN {X 0,Y 377.487,Z 681.49,A -85,B 0,C 180,E1 -12870.667,E2 -12870.667} C_VEL
LIN {X 0,Y 379.086,Z 668.048,A -85,B 0,C 180,E1 -12871.86,E2 -12871.86} C_VEL
LIN {X 0,Y 380.487,Z 653.912,A -85,B 0,C 180,E1 -12872.865,E2 -12872.865} C_VEL
LIN {X 0,Y 381.735,Z 638.695,A -85,B 0,C 180,E1 -12873.695,E2 -12873.695} C_VEL
LIN {X 0,Y 382.687,Z 622.935,A -85,B 0,C 180,E1 -12874.312,E2 -12874.312} C_VEL
LIN {X 0,Y 383.281,Z 606.1,A -85,B 0,C 180,E1 -12874.728,E2 -12874.728} C_VEL
LIN {X 0,Y 382.819,Z 600.298,A -85,B 0,C 180,E1 -12874.882,E2 -12874.882} C_VEL
LIN {X 0,Y 378.071,Z 581.671,A -85,B 0,C 180,E1 -12875.626,E2 -12875.626} C_VEL
LIN {X 0,Y 377.665,Z 575.869,A -85,B 0,C 180,E1 -12875.78,E2 -12875.78} C_VEL
LIN {X 0,Y 379.836,Z 487.575,A -85,B 0,C 180,E1 -12877.502,E2 -12877.502} C_VEL
LIN {X 0,Y 370.182,Z 465.406,A -85,B 0,C 180,E1 -12878.81,E2 -12878.81} C_VEL
LIN {X 0,Y 363.413,Z 451.326,A -85,B 0,C 180,E1 -12879.748,E2 -12879.748} C_VEL
LIN {X 0,Y 361.982,Z 446.008,A -85,B 0,C 180,E1 -12881.196,E2 -12881.196} C_VEL
LIN {X 0,Y 361.967,Z 446.023,A -85,B 0,C 180,E1 -12884.621,E2 -12884.621} C_VEL
LIN {X 0,Y 361.965,Z 446.019,A -85,B 0,C 180,E1 -12888.099,E2 -12888.099} C_VEL
LIN {X 0,Y 361.902,Z 446.028,A -85,B 0,C 180,E1 -12891.653,E2 -12891.653} C_VEL
LIN {X 0,Y 361.932,Z 446.022,A -85,B 0,C 180,E1 -12895.29,E2 -12895.29} C_VEL
LIN {X 0,Y 361.926,Z 446.019,A -85,B 0,C 180,E1 -12897.778,E2 -12897.778} C_VEL
LIN {X 0,Y 361.85,Z 446.036,A -85,B 0,C 180,E1 -12901.285,E2 -12901.285} C_VEL
LIN {X 0,Y 361.858,Z 446.035,A -85,B 0,C 180,E1 -12904.28,E2 -12904.28} C_VEL
LIN {X 0,Y 361.868,Z 446.025,A -85,B 0,C 180,E1 -12907.223,E2 -12907.223} C_VEL
LIN {X 0,Y 361.858,Z 446.033,A -85,B 0,C 180,E1 -12910.759,E2 -12910.759} C_VEL
LIN {X 0,Y 361.821,Z 446.036,A -85,B 0,C 180,E1 -12914.368,E2 -12914.368} C_VEL
LIN {X 0,Y 361.858,Z 446.029,A -85,B 0,C 180,E1 -12917.564,E2 -12917.564} C_VEL
LIN {X 0,Y 361.877,Z 446.031,A -85,B 0,C 180,E1 -12920.972,E2 -12920.972} C_VEL
LIN {X 0,Y 361.877,Z 446.022,A -85,B 0,C 180,E1 -12924.655,E2 -12924.655} C_VEL
LIN {X 0,Y 361.841,Z 446.032,A -85,B 0,C 180,E1 -12928.371,E2 -12928.371} C_VEL
LIN {X 0,Y 361.91,Z 446.027,A -85,B 0,C 180,E1 -12932.221,E2 -12932.221} C_VEL
LIN {X 0,Y 361.928,Z 446.022,A -85,B 0,C 180,E1 -12934.71,E2 -12934.71} C_VEL
LIN {X 0,Y 361.882,Z 446.028,A -85,B 0,C 180,E1 -12938.346,E2 -12938.346} C_VEL
LIN {X 0,Y 361.968,Z 446.011,A -85,B 0,C 180,E1 -12942.061,E2 -12942.061} C_VEL
LIN {X 0,Y 361.999,Z 446.017,A -85,B 0,C 180,E1 -12946.101,E2 -12946.101} C_VEL
LIN {X 0,Y 362.032,Z 445.998,A -85,B 0,C 180,E1 -12949.938,E2 -12949.938} C_VEL
LIN {X 0,Y 362.152,Z 445.996,A -85,B 0,C 180,E1 -12952.192,E2 -12952.192} C_VEL
LIN {X 0,Y 362.119,Z 445.999,A -85,B 0,C 180,E1 -12954.431,E2 -12954.431} C_VEL
LIN {X 0,Y 362.281,Z 445.97,A -85,B 0,C 180,E1 -12957.776,E2 -12957.776} C_VEL
LIN {X 0,Y 362.428,Z 445.965,A -85,B 0,C 180,E1 -12960,E2 -12960} C_VEL
LIN {X 0,Y 362.283,Z 445.975,A -85,B 0,C 180,E1 -12962.223,E2 -12962.223} C_VEL
LIN {X 0,Y 362.172,Z 445.989,A -85,B 0,C 180,E1 -12966.686,E2 -12966.686} C_VEL
LIN {X 0,Y 362.074,Z 446.006,A -85,B 0,C 180,E1 -12968.933,E2 -12968.933} C_VEL
LIN {X 0,Y 361.959,Z 446.006,A -85,B 0,C 180,E1 -12972.332,E2 -12972.332} C_VEL
LIN {X 0,Y 361.962,Z 446.019,A -85,B 0,C 180,E1 -12974.62,E2 -12974.62} C_VEL
LIN {X 0,Y 361.956,Z 446.007,A -85,B 0,C 180,E1 -12978.099,E2 -12978.099} C_VEL
LIN {X 0,Y 361.892,Z 446.034,A -85,B 0,C 180,E1 -12981.653,E2 -12981.653} C_VEL
LIN {X 0,Y 361.928,Z 446.027,A -85,B 0,C 180,E1 -12985.29,E2 -12985.29} C_VEL
LIN {X 0,Y 361.922,Z 446.027,A -85,B 0,C 180,E1 -12987.778,E2 -12987.778} C_VEL
LIN {X 0,Y 361.847,Z 446.034,A -85,B 0,C 180,E1 -12991.285,E2 -12991.285} C_VEL
LIN {X 0,Y 361.855,Z 446.035,A -85,B 0,C 180,E1 -12994.28,E2 -12994.28} C_VEL
LIN {X 0,Y 361.871,Z 446.034,A -85,B 0,C 180,E1 -12997.224,E2 -12997.224} C_VEL
LIN {X 0,Y 361.836,Z 446.036,A -85,B 0,C 180,E1 -13000.755,E2 -13000.755} C_VEL
LIN {X 0,Y 361.846,Z 446.035,A -85,B 0,C 180,E1 -13004.364,E2 -13004.364} C_VEL
LIN {X 0,Y 361.883,Z 446.033,A -85,B 0,C 180,E1 -13007.56,E2 -13007.56} C_VEL
LIN {X 0,Y 361.871,Z 446.034,A -85,B 0,C 180,E1 -13010.973,E2 -13010.973} C_VEL
LIN {X 0,Y 361.887,Z 446.133,A -85,B 0,C 180,E1 -13013.171,E2 -13013.171} C_VEL
LIN {X 0,Y 365.543,Z 459.758,A -85,B 0,C 180,E1 -13016.444,E2 -13016.444} C_VEL
LIN {X 0,Y 368.044,Z 469.899,A -85,B 0,C 180,E1 -13018.71,E2 -13018.71} C_VEL
LIN {X 0,Y 374.403,Z 484.982,A -85,B 0,C 180,E1 -13019.599,E2 -13019.599} C_VEL
LIN {X 0,Y 379.492,Z 512.158,A -85,B 0,C 180,E1 -13020.611,E2 -13020.611} C_VEL
LIN {X 0,Y 376.363,Z 635.839,A -85,B 0,C 180,E1 -13023.037,E2 -13023.037} C_VEL
LIN {X 0,Y 375.387,Z 652.033,A -85,B 0,C 180,E1 -13023.561,E2 -13023.561} C_VEL
LIN {X 0,Y 374.277,Z 665.459,A -85,B 0,C 180,E1 -13024.189,E2 -13024.189} C_VEL
LIN {X 0,Y 372.819,Z 679.711,A -85,B 0,C 180,E1 -13025.06,E2 -13025.06} C_VEL
LIN {X 0,Y 371.196,Z 693.415,A -85,B 0,C 180,E1 -13026.127,E2 -13026.127} C_VEL
LIN {X 0,Y 369.521,Z 706.09,A -85,B 0,C 180,E1 -13027.347,E2 -13027.347} C_VEL
LIN {X 0,Y 367.829,Z 717.856,A -85,B 0,C 180,E1 -13028.713,E2 -13028.713} C_VEL
LIN {X 0,Y 366.232,Z 728.905,A -85,B 0,C 180,E1 -13030.249,E2 -13030.249} C_VEL
LIN {X 0,Y 364.949,Z 738.144,A -85,B 0,C 180,E1 -13031.763,E2 -13031.763} C_VEL
LIN {X 0,Y 363.435,Z 748.139,A -85,B 0,C 180,E1 -13033.716,E2 -13033.716} C_VEL
LIN {X 0,Y 362.214,Z 757.06,A -85,B 0,C 180,E1 -13035.839,E2 -13035.839} C_VEL
LIN {X 0,Y 361.341,Z 765.074,A -85,B 0,C 180,E1 -13038.216,E2 -13038.216} C_VEL
LIN {X 0,Y 360.741,Z 771.084,A -85,B 0,C 180,E1 -13040.468,E2 -13040.468} C_VEL
LIN {X 0,Y 360.5,Z 774.64,A -85,B 0,C 180,E1 -13042.156,E2 -13042.156} C_VEL
LIN {X 0,Y 360.332,Z 778.27,A -85,B 0,C 180,E1 -13044.403,E2 -13044.403} C_VEL
LIN {X 0,Y 360.273,Z 780.672,A -85,B 0,C 180,E1 -13046.644,E2 -13046.644} C_VEL
LIN {X 0,Y 360.313,Z 781.9,A -85,B 0,C 180,E1 -13048.882,E2 -13048.882} C_VEL
LIN {X 0,Y 360.313,Z 781.917,A -85,B 0,C 180,E1 -13051.117,E2 -13051.117} C_VEL
LIN {X 0,Y 360.28,Z 780.777,A -85,B 0,C 180,E1 -13053.354,E2 -13053.354} C_VEL
LIN {X 0,Y 360.331,Z 778.478,A -85,B 0,C 180,E1 -13055.596,E2 -13055.596} C_VEL
LIN {X 0,Y 360.514,Z 774.972,A -85,B 0,C 180,E1 -13057.842,E2 -13057.842} C_VEL
LIN {X 0,Y 360.841,Z 770.174,A -85,B 0,C 180,E1 -13060.095,E2 -13060.095} C_VEL
LIN {X 0,Y 361.549,Z 763.959,A -85,B 0,C 180,E1 -13062.346,E2 -13062.346} C_VEL
LIN {X 0,Y 362.494,Z 756.154,A -85,B 0,C 180,E1 -13064.598,E2 -13064.598} C_VEL
LIN {X 0,Y 363.681,Z 747.856,A -85,B 0,C 180,E1 -13066.56,E2 -13066.56} C_VEL
LIN {X 0,Y 365.27,Z 737.893,A -85,B 0,C 180,E1 -13068.509,E2 -13068.509} C_VEL
LIN {X 0,Y 366.824,Z 727.696,A -85,B 0,C 180,E1 -13070.173,E2 -13070.173} C_VEL
LIN {X 0,Y 368.492,Z 716.671,A -85,B 0,C 180,E1 -13071.685,E2 -13071.685} C_VEL
LIN {X 0,Y 370.261,Z 704.797,A -85,B 0,C 180,E1 -13073.046,E2 -13073.046} C_VEL
LIN {X 0,Y 372.041,Z 691.981,A -85,B 0,C 180,E1 -13074.258,E2 -13074.258} C_VEL
LIN {X 0,Y 373.695,Z 678.323,A -85,B 0,C 180,E1 -13075.307,E2 -13075.307} C_VEL
LIN {X 0,Y 375.12,Z 664.545,A -85,B 0,C 180,E1 -13076.143,E2 -13076.143} C_VEL
LIN {X 0,Y 376.442,Z 649.871,A -85,B 0,C 180,E1 -13076.806,E2 -13076.806} C_VEL
LIN {X 0,Y 377.293,Z 635.596,A -85,B 0,C 180,E1 -13077.265,E2 -13077.265} C_VEL
LIN {X 0,Y 380.072,Z 534.647,A -85,B 0,C 180,E1 -13079.261,E2 -13079.261} C_VEL
